LIN {X 0,Y 491.211,Z 1235.46,A -85,B 0,C 180,E1 12597.361,E2 12597.361} C_VEL
LIN {X 0,Y 492.197,Z 1227.239,A -85,B 0,C 180,E1 12605.326,E2 12605.326} C_VEL
LIN {X 0,Y 494.194,Z 1205.404,A -85,B 0,C 180,E1 12612.883,E2 12612.883} C_VEL
LIN {X 0,Y 499.705,Z 1169.344,A -85,B 0,C 180,E1 12619.985,E2 12619.985} C_VEL
LIN {X 0,Y 507.992,Z 1121.366,A -85,B 0,C 180,E1 12625.908,E2 12625.908} C_VEL
LIN {X 0,Y 516.438,Z 1064.19,A -85,B 0,C 180,E1 12630.398,E2 12630.398} C_VEL
LIN {X 0,Y 519.366,Z 1023.748,A -85,B 0,C 180,E1 12632.582,E2 12632.582} C_VEL
LIN {X 0,Y 493.539,Z 958.868,A -85,B 0,C 180,E1 12636.637,E2 12636.637} C_VEL
LIN {X 0,Y 489.609,Z 948.94,A -85,B 0,C 180,E1 12637.215,E2 12637.215} C_VEL
LIN {X 0,Y 489.5,Z 948.94,A -85,B 0,C 180,E1 12646.8,E2 12646.8} C_VEL
LIN {X 0,Y 489.694,Z 948.94,A -85,B 0,C 180,E1 12657.113,E2 12657.113} C_VEL
LIN {X 0,Y 490.223,Z 950.204,A -85,B 0,C 180,E1 12666.559,E2 12666.559} C_VEL
LIN {X 0,Y 504.518,Z 1001.153,A -85,B 0,C 180,E1 12668.035,E2 12668.035} C_VEL
LIN {X 0,Y 503.347,Z 1055.895,A -85,B 0,C 180,E1 12669.439,E2 12669.439} C_VEL
LIN {X 0,Y 500.138,Z 1101.192,A -85,B 0,C 180,E1 12672.409,E2 12672.409} C_VEL
LIN {X 0,Y 496.485,Z 1136.434,A -85,B 0,C 180,E1 12676.706,E2 12676.706} C_VEL
LIN {X 0,Y 493.765,Z 1159.555,A -85,B 0,C 180,E1 12682.008,E2 12682.008} C_VEL
LIN {X 0,Y 492.775,Z 1168.783,A -85,B 0,C 180,E1 12687.309,E2 12687.309} C_VEL
LIN {X 0,Y 492.851,Z 1166.502,A -85,B 0,C 180,E1 12692.603,E2 12692.603} C_VEL
LIN {X 0,Y 494.456,Z 1150.28,A -85,B 0,C 180,E1 12698.337,E2 12698.337} C_VEL
LIN {X 0,Y 497.549,Z 1121.567,A -85,B 0,C 180,E1 12703.177,E2 12703.177} C_VEL
LIN {X 0,Y 501.349,Z 1080.414,A -85,B 0,C 180,E1 12706.955,E2 12706.955} C_VEL
LIN {X 0,Y 503.697,Z 1033.18,A -85,B 0,C 180,E1 12709.116,E2 12709.116} C_VEL
LIN {X 0,Y 501.948,Z 988.132,A -85,B 0,C 180,E1 12709.997,E2 12709.997} C_VEL
LIN {X 0,Y 490.032,Z 948.94,A -85,B 0,C 180,E1 12711.337,E2 12711.337} C_VEL
LIN {X 0,Y 489.534,Z 948.94,A -85,B 0,C 180,E1 12721.467,E2 12721.467} C_VEL
LIN {X 0,Y 489.452,Z 948.94,A -85,B 0,C 180,E1 12731.738,E2 12731.738} C_VEL
LIN {X 0,Y 489.581,Z 948.94,A -85,B 0,C 180,E1 12740.517,E2 12740.517} C_VEL
LIN {X 0,Y 489.797,Z 948.94,A -85,B 0,C 180,E1 12749.229,E2 12749.229} C_VEL
LIN {X 0,Y 490.061,Z 948.94,A -85,B 0,C 180,E1 12759.116,E2 12759.116} C_VEL
LIN {X 0,Y 490.905,Z 948.94,A -85,B 0,C 180,E1 12768.389,E2 12768.389} C_VEL
LIN {X 0,Y 490.724,Z 948.94,A -85,B 0,C 180,E1 12779.097,E2 12779.097} C_VEL
LIN {X 0,Y 490.401,Z 948.94,A -85,B 0,C 180,E1 12787.988,E2 12787.988} C_VEL
LIN {X 0,Y 489.983,Z 948.94,A -85,B 0,C 180,E1 12797.096,E2 12797.096} C_VEL
LIN {X 0,Y 489.779,Z 948.94,A -85,B 0,C 180,E1 12806.682,E2 12806.682} C_VEL
LIN {X 0,Y 489.937,Z 948.94,A -85,B 0,C 180,E1 12814.947,E2 12814.947} C_VEL
LIN {X 0,Y 489.655,Z 948.94,A -85,B 0,C 180,E1 12824.198,E2 12824.198} C_VEL
LIN {X 0,Y 489.798,Z 950.405,A -85,B 0,C 180,E1 12826.839,E2 12826.839} C_VEL
LIN {X 0,Y 518.54,Z 1013.899,A -85,B 0,C 180,E1 12831.17,E2 12831.17} C_VEL
LIN {X 0,Y 525.213,Z 1042.25,A -85,B 0,C 180,E1 12832.797,E2 12832.797} C_VEL
LIN {X 0,Y 514.365,Z 1115.654,A -85,B 0,C 180,E1 12836.471,E2 12836.471} C_VEL
LIN {X 0,Y 504.365,Z 1179.97,A -85,B 0,C 180,E1 12841.767,E2 12841.767} C_VEL
LIN {X 0,Y 497.073,Z 1230.999,A -85,B 0,C 180,E1 12848.228,E2 12848.228} C_VEL
LIN {X 0,Y 492.921,Z 1267.707,A -85,B 0,C 180,E1 12855.512,E2 12855.512} C_VEL
LIN {X 0,Y 491.499,Z 1286.659,A -85,B 0,C 180,E1 12862.006,E2 12862.006} C_VEL
LIN {X 0,Y 483.413,Z 1292.195,A -85,B 0,C 180,E1 12866.028,E2 12866.028} C_VEL
LIN {X 0,Y 483.428,Z 1292.84,A -85,B 0,C 180,E1 12872.743,E2 12872.743} C_VEL
LIN {X 0,Y 483.602,Z 1280.706,A -85,B 0,C 180,E1 12879.619,E2 12879.619} C_VEL
LIN {X 0,Y 485.229,Z 1255.323,A -85,B 0,C 180,E1 12886.158,E2 12886.158} C_VEL
LIN {X 0,Y 488.81,Z 1214.714,A -85,B 0,C 180,E1 12892.396,E2 12892.396} C_VEL
LIN {X 0,Y 494.43,Z 1155.575,A -85,B 0,C 180,E1 12898.201,E2 12898.201} C_VEL
LIN {X 0,Y 502.044,Z 1074.735,A -85,B 0,C 180,E1 12903.395,E2 12903.395} C_VEL
LIN {X 0,Y 506.039,Z 1025.461,A -85,B 0,C 180,E1 12905.719,E2 12905.719} C_VEL
LIN {X 0,Y 497.61,Z 982.294,A -85,B 0,C 180,E1 12908.629,E2 12908.629} C_VEL
LIN {X 0,Y 488.368,Z 961.377,A -85,B 0,C 180,E1 12911.493,E2 12911.493} C_VEL
LIN {X 0,Y 485.546,Z 955.861,A -85,B 0,C 180,E1 12913.699,E2 12913.699} C_VEL
LIN {X 0,Y 487.532,Z 959.576,A -85,B 0,C 180,E1 12915.666,E2 12915.666} C_VEL
LIN {X 0,Y 497.122,Z 976.809,A -85,B 0,C 180,E1 12918.204,E2 12918.204} C_VEL
LIN {X 0,Y 509.017,Z 1015.646,A -85,B 0,C 180,E1 12920.57,E2 12920.57} C_VEL
LIN {X 0,Y 511.87,Z 1042.243,A -85,B 0,C 180,E1 12921.963,E2 12921.963} C_VEL
LIN {X 0,Y 505.638,Z 1098.199,A -85,B 0,C 180,E1 12925.235,E2 12925.235} C_VEL
LIN {X 0,Y 497.291,Z 1149.138,A -85,B 0,C 180,E1 12930.205,E2 12930.205} C_VEL
LIN {X 0,Y 489.898,Z 1189.814,A -85,B 0,C 180,E1 12936.565,E2 12936.565} C_VEL
LIN {X 0,Y 485.077,Z 1218.909,A -85,B 0,C 180,E1 12944.128,E2 12944.128} C_VEL
LIN {X 0,Y 483.428,Z 1233.639,A -85,B 0,C 180,E1 12951.896,E2 12951.896} C_VEL
LIN {X 0,Y 483.632,Z 1235.321,A -85,B 0,C 180,E1 12959.119,E2 12959.119} C_VEL
LIN {X 0,Y 484.255,Z 1225.816,A -85,B 0,C 180,E1 12966.316,E2 12966.316} C_VEL
LIN {X 0,Y 486.687,Z 1202.499,A -85,B 0,C 180,E1 12973.931,E2 12973.931} C_VEL
LIN {X 0,Y 492.837,Z 1165.138,A -85,B 0,C 180,E1 12980.997,E2 12980.997} C_VEL
LIN {X 0,Y 501.852,Z 1114.197,A -85,B 0,C 180,E1 12987.015,E2 12987.015} C_VEL
LIN {X 0,Y 510.637,Z 1055.281,A -85,B 0,C 180,E1 12991.363,E2 12991.363} C_VEL
LIN {X 0,Y 512.254,Z 1026.098,A -85,B 0,C 180,E1 12992.931,E2 12992.931} C_VEL
LIN {X 0,Y 486.656,Z 961.716,A -85,B 0,C 180,E1 12997.077,E2 12997.077} C_VEL
LIN {X 0,Y 481.499,Z 948.94,A -85,B 0,C 180,E1 12997.952,E2 12997.952} C_VEL
LIN {X 0,Y 481.524,Z 948.94,A -85,B 0,C 180,E1 13007.821,E2 13007.821} C_VEL
LIN {X 0,Y 481.663,Z 948.94,A -85,B 0,C 180,E1 13016.654,E2 13016.654} C_VEL
LIN {X 0,Y 482.137,Z 950.075,A -85,B 0,C 180,E1 13026.137,E2 13026.137} C_VEL
LIN {X 0,Y 497.113,Z 1003.116,A -85,B 0,C 180,E1 13027.718,E2 13027.718} C_VEL
LIN {X 0,Y 495.929,Z 1056.161,A -85,B 0,C 180,E1 13029.097,E2 13029.097} C_VEL
LIN {X 0,Y 492.737,Z 1100.792,A -85,B 0,C 180,E1 13032.02,E2 13032.02} C_VEL
LIN {X 0,Y 488.965,Z 1135.924,A -85,B 0,C 180,E1 13036.269,E2 13036.269} C_VEL
LIN {X 0,Y 486.183,Z 1159.161,A -85,B 0,C 180,E1 13041.431,E2 13041.431} C_VEL
LIN {X 0,Y 484.857,Z 1169.728,A -85,B 0,C 180,E1 13047.265,E2 13047.265} C_VEL
LIN {X 0,Y 484.934,Z 1167.468,A -85,B 0,C 180,E1 13052.646,E2 13052.646} C_VEL
LIN {X 0,Y 486.608,Z 1151.273,A -85,B 0,C 180,E1 13058.473,E2 13058.473} C_VEL
LIN {X 0,Y 489.828,Z 1122.592,A -85,B 0,C 180,E1 13063.388,E2 13063.388} C_VEL
LIN {X 0,Y 493.774,Z 1081.501,A -85,B 0,C 180,E1 13067.223,E2 13067.223} C_VEL
LIN {X 0,Y 496.241,Z 1033.419,A -85,B 0,C 180,E1 13069.445,E2 13069.445} C_VEL
LIN {X 0,Y 494.378,Z 989.209,A -85,B 0,C 180,E1 13070.324,E2 13070.324} C_VEL
LIN {X 0,Y 481.964,Z 948.94,A -85,B 0,C 180,E1 13071.67,E2 13071.67} C_VEL
LIN {X 0,Y 481.548,Z 948.94,A -85,B 0,C 180,E1 13081.272,E2 13081.272} C_VEL
LIN {X 0,Y 481.381,Z 948.94,A -85,B 0,C 180,E1 13090.193,E2 13090.193} C_VEL
LIN {X 0,Y 481.588,Z 948.94,A -85,B 0,C 180,E1 13100.453,E2 13100.453} C_VEL
LIN {X 0,Y 481.781,Z 948.94,A -85,B 0,C 180,E1 13110.75,E2 13110.75} C_VEL
LIN {X 0,Y 482.133,Z 948.94,A -85,B 0,C 180,E1 13120.679,E2 13120.679} C_VEL
LIN {X 0,Y 482.743,Z 948.94,A -85,B 0,C 180,E1 13130.024,E2 13130.024} C_VEL
LIN {X 0,Y 482.726,Z 948.94,A -85,B 0,C 180,E1 13139.082,E2 13139.082} C_VEL
LIN {X 0,Y 482.403,Z 948.94,A -85,B 0,C 180,E1 13148.122,E2 13148.122} C_VEL
LIN {X 0,Y 481.977,Z 948.94,A -85,B 0,C 180,E1 13157.389,E2 13157.389} C_VEL
LIN {X 0,Y 481.8,Z 948.94,A -85,B 0,C 180,E1 13167.16,E2 13167.16} C_VEL
LIN {X 0,Y 481.789,Z 948.94,A -85,B 0,C 180,E1 13176.652,E2 13176.652} C_VEL
LIN {X 0,Y 481.839,Z 950.706,A -85,B 0,C 180,E1 13186.117,E2 13186.117} C_VEL
LIN {X 0,Y 511.726,Z 1016.286,A -85,B 0,C 180,E1 13190.757,E2 13190.757} C_VEL
LIN {X 0,Y 518.055,Z 1044.204,A -85,B 0,C 180,E1 13192.418,E2 13192.418} C_VEL
LIN {X 0,Y 506.873,Z 1117.207,A -85,B 0,C 180,E1 13196.187,E2 13196.187} C_VEL
LIN {X 0,Y 496.491,Z 1181.713,A -85,B 0,C 180,E1 13201.66,E2 13201.66} C_VEL
LIN {X 0,Y 488.937,Z 1232.789,A -85,B 0,C 180,E1 13208.342,E2 13208.342} C_VEL
LIN {X 0,Y 484.766,Z 1268.623,A -85,B 0,C 180,E1 13215.741,E2 13215.741} C_VEL
LIN {X 0,Y 483.351,Z 1287.892,A -85,B 0,C 180,E1 13222.832,E2 13222.832} C_VEL
LIN {X 0,Y 483.413,Z 1292.195,A -85,B 0,C 180,E1 13226.028,E2 13226.028} C_VEL
LIN {X 0,Y 475.431,Z 1293.448,A -85,B 0,C 180,E1 13230.149,E2 13230.149} C_VEL
LIN {X 0,Y 475.669,Z 1285.828,A -85,B 0,C 180,E1 13237.376,E2 13237.376} C_VEL
LIN {X 0,Y 476.612,Z 1264.154,A -85,B 0,C 180,E1 13244.33,E2 13244.33} C_VEL
LIN {X 0,Y 479.603,Z 1228.689,A -85,B 0,C 180,E1 13250.722,E2 13250.722} C_VEL
LIN {X 0,Y 484.576,Z 1177.402,A -85,B 0,C 180,E1 13256.609,E2 13256.609} C_VEL
LIN {X 0,Y 492.062,Z 1103.72,A -85,B 0,C 180,E1 13262.17,E2 13262.17} C_VEL
LIN {X 0,Y 499.161,Z 1027.522,A -85,B 0,C 180,E1 13266.155,E2 13266.155} C_VEL
LIN {X 0,Y 492.068,Z 986.499,A -85,B 0,C 180,E1 13269.1,E2 13269.1} C_VEL
LIN {X 0,Y 484.839,Z 968.073,A -85,B 0,C 180,E1 13271.826,E2 13271.826} C_VEL
LIN {X 0,Y 483.253,Z 963.504,A -85,B 0,C 180,E1 13273.699,E2 13273.699} C_VEL
LIN {X 0,Y 485.534,Z 968.12,A -85,B 0,C 180,E1 13275.738,E2 13275.738} C_VEL
LIN {X 0,Y 494.868,Z 987.686,A -85,B 0,C 180,E1 13278.238,E2 13278.238} C_VEL
LIN {X 0,Y 505.961,Z 1038.4,A -85,B 0,C 180,E1 13281.22,E2 13281.22} C_VEL
LIN {X 0,Y 499.43,Z 1095.926,A -85,B 0,C 180,E1 13284.484,E2 13284.484} C_VEL
LIN {X 0,Y 490.562,Z 1148.251,A -85,B 0,C 180,E1 13289.555,E2 13289.555} C_VEL
LIN {X 0,Y 482.664,Z 1189.461,A -85,B 0,C 180,E1 13296.001,E2 13296.001} C_VEL
LIN {X 0,Y 477.603,Z 1218.168,A -85,B 0,C 180,E1 13303.399,E2 13303.399} C_VEL
LIN {X 0,Y 475.561,Z 1233.069,A -85,B 0,C 180,E1 13310.836,E2 13310.836} C_VEL
LIN {X 0,Y 475.656,Z 1235.818,A -85,B 0,C 180,E1 13319.104,E2 13319.104} C_VEL
LIN {X 0,Y 476.291,Z 1226.268,A -85,B 0,C 180,E1 13326.422,E2 13326.422} C_VEL
LIN {X 0,Y 478.805,Z 1203.262,A -85,B 0,C 180,E1 13334.059,E2 13334.059} C_VEL
LIN {X 0,Y 485.043,Z 1166.834,A -85,B 0,C 180,E1 13341.11,E2 13341.11} C_VEL
LIN {X 0,Y 494.309,Z 1116.083,A -85,B 0,C 180,E1 13347.252,E2 13347.252} C_VEL
LIN {X 0,Y 503.468,Z 1056.622,A -85,B 0,C 180,E1 13351.734,E2 13351.734} C_VEL
LIN {X 0,Y 504.78,Z 1027.337,A -85,B 0,C 180,E1 13353.364,E2 13353.364} C_VEL
LIN {X 0,Y 479.243,Z 962.842,A -85,B 0,C 180,E1 13357.605,E2 13357.605} C_VEL
LIN {X 0,Y 473.422,Z 948.94,A -85,B 0,C 180,E1 13358.489,E2 13358.489} C_VEL
LIN {X 0,Y 473.478,Z 948.94,A -85,B 0,C 180,E1 13368.907,E2 13368.907} C_VEL
LIN {X 0,Y 473.668,Z 948.94,A -85,B 0,C 180,E1 13378.154,E2 13378.154} C_VEL
LIN {X 0,Y 474.094,Z 950.032,A -85,B 0,C 180,E1 13385.703,E2 13385.703} C_VEL
LIN {X 0,Y 489.716,Z 1004.431,A -85,B 0,C 180,E1 13387.382,E2 13387.382} C_VEL
LIN {X 0,Y 488.405,Z 1058.374,A -85,B 0,C 180,E1 13388.833,E2 13388.833} C_VEL
LIN {X 0,Y 484.877,Z 1104.074,A -85,B 0,C 180,E1 13391.954,E2 13391.954} C_VEL
LIN {X 0,Y 480.827,Z 1139.501,A -85,B 0,C 180,E1 13396.497,E2 13396.497} C_VEL
LIN {X 0,Y 477.851,Z 1162.687,A -85,B 0,C 180,E1 13402.199,E2 13402.199} C_VEL
LIN {X 0,Y 476.943,Z 1170.672,A -85,B 0,C 180,E1 13407.22,E2 13407.22} C_VEL
LIN {X 0,Y 477.002,Z 1168.436,A -85,B 0,C 180,E1 13412.69,E2 13412.69} C_VEL
LIN {X 0,Y 478.771,Z 1152.266,A -85,B 0,C 180,E1 13418.612,E2 13418.612} C_VEL
LIN {X 0,Y 482.141,Z 1123.613,A -85,B 0,C 180,E1 13423.606,E2 13423.606} C_VEL
LIN {X 0,Y 486.231,Z 1082.61,A -85,B 0,C 180,E1 13427.497,E2 13427.497} C_VEL
LIN {X 0,Y 488.765,Z 1034.7,A -85,B 0,C 180,E1 13429.755,E2 13429.755} C_VEL
LIN {X 0,Y 486.955,Z 990.574,A -85,B 0,C 180,E1 13430.651,E2 13430.651} C_VEL
LIN {X 0,Y 473.877,Z 948.94,A -85,B 0,C 180,E1 13432.065,E2 13432.065} C_VEL
LIN {X 0,Y 473.483,Z 948.94,A -85,B 0,C 180,E1 13441.867,E2 13441.867} C_VEL
LIN {X 0,Y 473.35,Z 948.94,A -85,B 0,C 180,E1 13451.075,E2 13451.075} C_VEL
LIN {X 0,Y 473.552,Z 948.94,A -85,B 0,C 180,E1 13461.295,E2 13461.295} C_VEL
LIN {X 0,Y 473.738,Z 948.94,A -85,B 0,C 180,E1 13471.638,E2 13471.638} C_VEL
LIN {X 0,Y 474.228,Z 948.94,A -85,B 0,C 180,E1 13482.28,E2 13482.28} C_VEL
LIN {X 0,Y 474.739,Z 948.94,A -85,B 0,C 180,E1 13489.854,E2 13489.854} C_VEL
LIN {X 0,Y 474.729,Z 948.94,A -85,B 0,C 180,E1 13499.066,E2 13499.066} C_VEL
LIN {X 0,Y 474.38,Z 948.94,A -85,B 0,C 180,E1 13508.26,E2 13508.26} C_VEL
LIN {X 0,Y 473.937,Z 948.94,A -85,B 0,C 180,E1 13517.694,E2 13517.694} C_VEL
LIN {X 0,Y 473.793,Z 948.94,A -85,B 0,C 180,E1 13528.374,E2 13528.374} C_VEL
LIN {X 0,Y 473.776,Z 948.94,A -85,B 0,C 180,E1 13538.638,E2 13538.638} C_VEL
LIN {X 0,Y 473.693,Z 950.046,A -85,B 0,C 180,E1 13545.324,E2 13545.324} C_VEL
LIN {X 0,Y 504.735,Z 1018.436,A -85,B 0,C 180,E1 13550.321,E2 13550.321} C_VEL
LIN {X 0,Y 510.8,Z 1046.867,A -85,B 0,C 180,E1 13552.058,E2 13552.058} C_VEL
LIN {X 0,Y 499.452,Z 1117.969,A -85,B 0,C 180,E1 13555.857,E2 13555.857} C_VEL
LIN {X 0,Y 488.666,Z 1182.726,A -85,B 0,C 180,E1 13561.481,E2 13561.481} C_VEL
LIN {X 0,Y 480.986,Z 1233.279,A -85,B 0,C 180,E1 13568.256,E2 13568.256} C_VEL
LIN {X 0,Y 476.725,Z 1268.936,A -85,B 0,C 180,E1 13575.814,E2 13575.814} C_VEL
LIN {X 0,Y 475.384,Z 1287.302,A -85,B 0,C 180,E1 13582.711,E2 13582.711} C_VEL
LIN {X 0,Y 475.431,Z 1293.448,A -85,B 0,C 180,E1 13590.149,E2 13590.149} C_VEL
LIN {X 0,Y 467.315,Z 1290.285,A -85,B 0,C 180,E1 13594.35,E2 13594.35} C_VEL
LIN {X 0,Y 468.077,Z 1275.571,A -85,B 0,C 180,E1 13601.262,E2 13601.262} C_VEL
LIN {X 0,Y 470.614,Z 1244.576,A -85,B 0,C 180,E1 13608.369,E2 13608.369} C_VEL
LIN {X 0,Y 474.965,Z 1198.501,A -85,B 0,C 180,E1 13614.726,E2 13614.726} C_VEL
LIN {X 0,Y 481.596,Z 1133.866,A -85,B 0,C 180,E1 13620.543,E2 13620.543} C_VEL
LIN {X 0,Y 491.741,Z 1047.179,A -85,B 0,C 180,E1 13625.688,E2 13625.688} C_VEL
LIN {X 0,Y 491.841,Z 1025.815,A -85,B 0,C 180,E1 13626.899,E2 13626.899} C_VEL
LIN {X 0,Y 486.665,Z 990.335,A -85,B 0,C 180,E1 13629.65,E2 13629.65} C_VEL
LIN {X 0,Y 481.456,Z 974.599,A -85,B 0,C 180,E1 13632.223,E2 13632.223} C_VEL
LIN {X 0,Y 481.528,Z 971.562,A -85,B 0,C 180,E1 13634.562,E2 13634.562} C_VEL
LIN {X 0,Y 488.204,Z 987.393,A -85,B 0,C 180,E1 13637.276,E2 13637.276} C_VEL
LIN {X 0,Y 497.979,Z 1027.568,A -85,B 0,C 180,E1 13639.923,E2 13639.923} C_VEL
LIN {X 0,Y 498.576,Z 1052.151,A -85,B 0,C 180,E1 13641.223,E2 13641.223} C_VEL
LIN {X 0,Y 490.797,Z 1109.651,A -85,B 0,C 180,E1 13644.988,E2 13644.988} C_VEL
LIN {X 0,Y 481.538,Z 1158.317,A -85,B 0,C 180,E1 13650.292,E2 13650.292} C_VEL
LIN {X 0,Y 473.59,Z 1197.357,A -85,B 0,C 180,E1 13657.153,E2 13657.153} C_VEL
LIN {X 0,Y 468.851,Z 1223.639,A -85,B 0,C 180,E1 13665.009,E2 13665.009} C_VEL
LIN {X 0,Y 467.446,Z 1235.175,A -85,B 0,C 180,E1 13672.218,E2 13672.218} C_VEL
LIN {X 0,Y 467.659,Z 1236.315,A -85,B 0,C 180,E1 13679.088,E2 13679.088} C_VEL
LIN {X 0,Y 468.315,Z 1226.704,A -85,B 0,C 180,E1 13686.532,E2 13686.532} C_VEL
LIN {X 0,Y 470.986,Z 1203.576,A -85,B 0,C 180,E1 13694.297,E2 13694.297} C_VEL
LIN {X 0,Y 477.457,Z 1166.945,A -85,B 0,C 180,E1 13701.462,E2 13701.462} C_VEL
LIN {X 0,Y 487.048,Z 1116.162,A -85,B 0,C 180,E1 13707.663,E2 13707.663} C_VEL
LIN {X 0,Y 496.543,Z 1055.848,A -85,B 0,C 180,E1 13712.23,E2 13712.23} C_VEL
LIN {X 0,Y 497.927,Z 1030.54,A -85,B 0,C 180,E1 13713.661,E2 13713.661} C_VEL
LIN {X 0,Y 472.826,Z 966.515,A -85,B 0,C 180,E1 13718.003,E2 13718.003} C_VEL
LIN {X 0,Y 465.348,Z 948.94,A -85,B 0,C 180,E1 13719.074,E2 13719.074} C_VEL
LIN {X 0,Y 465.34,Z 948.94,A -85,B 0,C 180,E1 13727.993,E2 13727.993} C_VEL
LIN {X 0,Y 465.553,Z 948.94,A -85,B 0,C 180,E1 13737.415,E2 13737.415} C_VEL
LIN {X 0,Y 465.952,Z 949.108,A -85,B 0,C 180,E1 13745.232,E2 13745.232} C_VEL
LIN {X 0,Y 482.37,Z 1002.612,A -85,B 0,C 180,E1 13746.987,E2 13746.987} C_VEL
LIN {X 0,Y 481.055,Z 1058.272,A -85,B 0,C 180,E1 13748.454,E2 13748.454} C_VEL
LIN {X 0,Y 477.449,Z 1103.682,A -85,B 0,C 180,E1 13751.544,E2 13751.544} C_VEL
LIN {X 0,Y 473.333,Z 1139.095,A -85,B 0,C 180,E1 13756.042,E2 13756.042} C_VEL
LIN {X 0,Y 470.181,Z 1162.32,A -85,B 0,C 180,E1 13761.604,E2 13761.604} C_VEL
LIN {X 0,Y 469.025,Z 1171.617,A -85,B 0,C 180,E1 13767.173,E2 13767.173} C_VEL
LIN {X 0,Y 469.086,Z 1169.402,A -85,B 0,C 180,E1 13772.735,E2 13772.735} C_VEL
LIN {X 0,Y 470.946,Z 1153.257,A -85,B 0,C 180,E1 13778.757,E2 13778.757} C_VEL
LIN {X 0,Y 474.443,Z 1124.636,A -85,B 0,C 180,E1 13783.831,E2 13783.831} C_VEL
LIN {X 0,Y 478.687,Z 1083.694,A -85,B 0,C 180,E1 13787.782,E2 13787.782} C_VEL
LIN {X 0,Y 481.351,Z 1035.063,A -85,B 0,C 180,E1 13790.098,E2 13790.098} C_VEL
LIN {X 0,Y 479.674,Z 992.598,A -85,B 0,C 180,E1 13790.971,E2 13790.971} C_VEL
LIN {X 0,Y 465.838,Z 948.94,A -85,B 0,C 180,E1 13792.503,E2 13792.503} C_VEL
LIN {X 0,Y 465.388,Z 948.94,A -85,B 0,C 180,E1 13802.489,E2 13802.489} C_VEL
LIN {X 0,Y 465.323,Z 948.94,A -85,B 0,C 180,E1 13812.758,E2 13812.758} C_VEL
LIN {X 0,Y 465.521,Z 948.94,A -85,B 0,C 180,E1 13822.913,E2 13822.913} C_VEL
LIN {X 0,Y 465.751,Z 948.94,A -85,B 0,C 180,E1 13833.516,E2 13833.516} C_VEL
LIN {X 0,Y 466.428,Z 948.94,A -85,B 0,C 180,E1 13843.924,E2 13843.924} C_VEL
LIN {X 0,Y 466.414,Z 948.94,A -85,B 0,C 180,E1 13853.442,E2 13853.442} C_VEL
LIN {X 0,Y 466.568,Z 948.94,A -85,B 0,C 180,E1 13860.914,E2 13860.914} C_VEL
LIN {X 0,Y 466.293,Z 948.94,A -85,B 0,C 180,E1 13870.295,E2 13870.295} C_VEL
LIN {X 0,Y 465.85,Z 948.94,A -85,B 0,C 180,E1 13879.986,E2 13879.986} C_VEL
LIN {X 0,Y 465.812,Z 948.94,A -85,B 0,C 180,E1 13890.417,E2 13890.417} C_VEL
LIN {X 0,Y 465.612,Z 948.94,A -85,B 0,C 180,E1 13900.095,E2 13900.095} C_VEL
LIN {X 0,Y 465.859,Z 950.978,A -85,B 0,C 180,E1 13904.595,E2 13904.595} C_VEL
LIN {X 0,Y 497.47,Z 1019.856,A -85,B 0,C 180,E1 13909.836,E2 13909.836} C_VEL
LIN {X 0,Y 503.621,Z 1049.011,A -85,B 0,C 180,E1 13911.675,E2 13911.675} C_VEL
LIN {X 0,Y 491.73,Z 1120.498,A -85,B 0,C 180,E1 13915.648,E2 13915.648} C_VEL
LIN {X 0,Y 480.811,Z 1183.919,A -85,B 0,C 180,E1 13921.325,E2 13921.325} C_VEL
LIN {X 0,Y 472.99,Z 1234.05,A -85,B 0,C 180,E1 13928.227,E2 13928.227} C_VEL
LIN {X 0,Y 468.664,Z 1269.61,A -85,B 0,C 180,E1 13935.995,E2 13935.995} C_VEL
LIN {X 0,Y 467.324,Z 1288.245,A -85,B 0,C 180,E1 13943.521,E2 13943.521} C_VEL
LIN {X 0,Y 467.709,Z 1292.88,A -85,B 0,C 180,E1 13950.975,E2 13950.975} C_VEL
LIN {X 0,Y 467.315,Z 1290.285,A -85,B 0,C 180,E1 13954.35,E2 13954.35} C_VEL
LIN {X 0,Y 459.589,Z 1282.729,A -85,B 0,C 180,E1 13958.551,E2 13958.551} C_VEL
LIN {X 0,Y 460.933,Z 1259.457,A -85,B 0,C 180,E1 13965.561,E2 13965.561} C_VEL
LIN {X 0,Y 464.53,Z 1221.78,A -85,B 0,C 180,E1 13972.112,E2 13972.112} C_VEL
LIN {X 0,Y 470.574,Z 1165.89,A -85,B 0,C 180,E1 13978.318,E2 13978.318} C_VEL
LIN {X 0,Y 480.067,Z 1085.232,A -85,B 0,C 180,E1 13984.215,E2 13984.215} C_VEL
LIN {X 0,Y 485.802,Z 1030.749,A -85,B 0,C 180,E1 13987.213,E2 13987.213} C_VEL
LIN {X 0,Y 481.853,Z 995.487,A -85,B 0,C 180,E1 13990.092,E2 13990.092} C_VEL
LIN {X 0,Y 478.35,Z 979.934,A -85,B 0,C 180,E1 13993.058,E2 13993.058} C_VEL
LIN {X 0,Y 479.54,Z 981.557,A -85,B 0,C 180,E1 13994.971,E2 13994.971} C_VEL
LIN {X 0,Y 486.123,Z 999.348,A -85,B 0,C 180,E1 13997.4,E2 13997.4} C_VEL
LIN {X 0,Y 493.093,Z 1046.988,A -85,B 0,C 180,E1 14000.351,E2 14000.351} C_VEL
LIN {X 0,Y 485.494,Z 1103.489,A -85,B 0,C 180,E1 14003.858,E2 14003.858} C_VEL
LIN {X 0,Y 475.702,Z 1153.945,A -85,B 0,C 180,E1 14009.124,E2 14009.124} C_VEL
LIN {X 0,Y 467.052,Z 1193.721,A -85,B 0,C 180,E1 14015.824,E2 14015.824} C_VEL
LIN {X 0,Y 461.465,Z 1221.805,A -85,B 0,C 180,E1 14023.784,E2 14023.784} C_VEL
LIN {X 0,Y 459.577,Z 1235.227,A -85,B 0,C 180,E1 14031.472,E2 14031.472} C_VEL
LIN {X 0,Y 459.678,Z 1236.81,A -85,B 0,C 180,E1 14039.073,E2 14039.073} C_VEL
LIN {X 0,Y 460.372,Z 1226.184,A -85,B 0,C 180,E1 14047.121,E2 14047.121} C_VEL
LIN {X 0,Y 463.371,Z 1202.386,A -85,B 0,C 180,E1 14054.912,E2 14054.912} C_VEL
LIN {X 0,Y 470.154,Z 1165.495,A -85,B 0,C 180,E1 14062.054,E2 14062.054} C_VEL
LIN {X 0,Y 479.78,Z 1116.131,A -85,B 0,C 180,E1 14068.092,E2 14068.092} C_VEL
LIN {X 0,Y 489.396,Z 1056.98,A -85,B 0,C 180,E1 14072.627,E2 14072.627} C_VEL
LIN {X 0,Y 490.468,Z 1032.092,A -85,B 0,C 180,E1 14074.087,E2 14074.087} C_VEL
LIN {X 0,Y 465.279,Z 967.484,A -85,B 0,C 180,E1 14078.562,E2 14078.562} C_VEL
LIN {X 0,Y 457.271,Z 948.94,A -85,B 0,C 180,E1 14079.935,E2 14079.935} C_VEL
LIN {X 0,Y 457.359,Z 948.94,A -85,B 0,C 180,E1 14089.63,E2 14089.63} C_VEL
LIN {X 0,Y 457.55,Z 948.94,A -85,B 0,C 180,E1 14099.015,E2 14099.015} C_VEL
LIN {X 0,Y 457.993,Z 950.221,A -85,B 0,C 180,E1 14104.788,E2 14104.788} C_VEL
LIN {X 0,Y 475.014,Z 1003.297,A -85,B 0,C 180,E1 14106.618,E2 14106.618} C_VEL
LIN {X 0,Y 473.743,Z 1057.677,A -85,B 0,C 180,E1 14108.045,E2 14108.045} C_VEL
LIN {X 0,Y 470.114,Z 1103.282,A -85,B 0,C 180,E1 14111.123,E2 14111.123} C_VEL
LIN {X 0,Y 465.829,Z 1138.577,A -85,B 0,C 180,E1 14115.572,E2 14115.572} C_VEL
LIN {X 0,Y 462.617,Z 1161.99,A -85,B 0,C 180,E1 14121.015,E2 14121.015} C_VEL
LIN {X 0,Y 461.088,Z 1172.565,A -85,B 0,C 180,E1 14127.124,E2 14127.124} C_VEL
LIN {X 0,Y 461.182,Z 1170.365,A -85,B 0,C 180,E1 14132.782,E2 14132.782} C_VEL
LIN {X 0,Y 463.124,Z 1154.248,A -85,B 0,C 180,E1 14138.906,E2 14138.906} C_VEL
LIN {X 0,Y 466.772,Z 1125.656,A -85,B 0,C 180,E1 14144.063,E2 14144.063} C_VEL
LIN {X 0,Y 471.17,Z 1084.692,A -85,B 0,C 180,E1 14148.082,E2 14148.082} C_VEL
LIN {X 0,Y 473.921,Z 1036.351,A -85,B 0,C 180,E1 14150.427,E2 14150.427} C_VEL
LIN {X 0,Y 472.018,Z 993.132,A -85,B 0,C 180,E1 14151.345,E2 14151.345} C_VEL
LIN {X 0,Y 457.779,Z 948.94,A -85,B 0,C 180,E1 14152.955,E2 14152.955} C_VEL
LIN {X 0,Y 457.349,Z 948.94,A -85,B 0,C 180,E1 14163.132,E2 14163.132} C_VEL
LIN {X 0,Y 457.328,Z 948.94,A -85,B 0,C 180,E1 14172.789,E2 14172.789} C_VEL
LIN {X 0,Y 457.413,Z 948.94,A -85,B 0,C 180,E1 14182.106,E2 14182.106} C_VEL
LIN {X 0,Y 457.704,Z 948.94,A -85,B 0,C 180,E1 14191.359,E2 14191.359} C_VEL
LIN {X 0,Y 458.112,Z 948.94,A -85,B 0,C 180,E1 14201.635,E2 14201.635} C_VEL
LIN {X 0,Y 458.742,Z 948.94,A -85,B 0,C 180,E1 14209.496,E2 14209.496} C_VEL
LIN {X 0,Y 458.733,Z 948.94,A -85,B 0,C 180,E1 14219.034,E2 14219.034} C_VEL
LIN {X 0,Y 458.36,Z 948.94,A -85,B 0,C 180,E1 14228.551,E2 14228.551} C_VEL
LIN {X 0,Y 457.861,Z 948.94,A -85,B 0,C 180,E1 14238.337,E2 14238.337} C_VEL
LIN {X 0,Y 457.747,Z 948.94,A -85,B 0,C 180,E1 14248.716,E2 14248.716} C_VEL
LIN {X 0,Y 457.621,Z 948.94,A -85,B 0,C 180,E1 14258.892,E2 14258.892} C_VEL
LIN {X 0,Y 457.651,Z 950.426,A -85,B 0,C 180,E1 14263.761,E2 14263.761} C_VEL
LIN {X 0,Y 490.563,Z 1022.424,A -85,B 0,C 180,E1 14269.434,E2 14269.434} C_VEL
LIN {X 0,Y 496.519,Z 1050.691,A -85,B 0,C 180,E1 14271.267,E2 14271.267} C_VEL
LIN {X 0,Y 483.695,Z 1124.469,A -85,B 0,C 180,E1 14275.541,E2 14275.541} C_VEL
LIN {X 0,Y 472.63,Z 1187.1,A -85,B 0,C 180,E1 14281.397,E2 14281.397} C_VEL
LIN {X 0,Y 464.713,Z 1237.124,A -85,B 0,C 180,E1 14288.611,E2 14288.611} C_VEL
LIN {X 0,Y 460.472,Z 1270.969,A -85,B 0,C 180,E1 14296.423,E2 14296.423} C_VEL
LIN {X 0,Y 459.348,Z 1287.63,A -85,B 0,C 180,E1 14303.408,E2 14303.408} C_VEL
LIN {X 0,Y 459.723,Z 1292.376,A -85,B 0,C 180,E1 14310.992,E2 14310.992} C_VEL
LIN {X 0,Y 459.589,Z 1282.729,A -85,B 0,C 180,E1 14318.551,E2 14318.551} C_VEL
LIN {X 0,Y 452.516,Z 1271.023,A -85,B 0,C 180,E1 14322.678,E2 14322.678} C_VEL
LIN {X 0,Y 455.306,Z 1238.488,A -85,B 0,C 180,E1 14329.769,E2 14329.769} C_VEL
LIN {X 0,Y 460.577,Z 1189.684,A -85,B 0,C 180,E1 14336.313,E2 14336.313} C_VEL
LIN {X 0,Y 468.93,Z 1119.675,A -85,B 0,C 180,E1 14342.47,E2 14342.47} C_VEL
LIN {X 0,Y 479.653,Z 1033.664,A -85,B 0,C 180,E1 14347.711,E2 14347.711} C_VEL
LIN {X 0,Y 477.079,Z 999.349,A -85,B 0,C 180,E1 14350.749,E2 14350.749} C_VEL
LIN {X 0,Y 475.851,Z 987.226,A -85,B 0,C 180,E1 14353.34,E2 14353.34} C_VEL
LIN {X 0,Y 477.82,Z 991.282,A -85,B 0,C 180,E1 14355.305,E2 14355.305} C_VEL
LIN {X 0,Y 484.183,Z 1015.954,A -85,B 0,C 180,E1 14357.729,E2 14357.729} C_VEL
LIN {X 0,Y 486.779,Z 1052.082,A -85,B 0,C 180,E1 14359.92,E2 14359.92} C_VEL
LIN {X 0,Y 478.306,Z 1109.067,A -85,B 0,C 180,E1 14363.665,E2 14363.665} C_VEL
LIN {X 0,Y 467.716,Z 1159.37,A -85,B 0,C 180,E1 14369.226,E2 14369.226} C_VEL
LIN {X 0,Y 458.607,Z 1198.714,A -85,B 0,C 180,E1 14376.361,E2 14376.361} C_VEL
LIN {X 0,Y 453.182,Z 1224.837,A -85,B 0,C 180,E1 14384.478,E2 14384.478} C_VEL
LIN {X 0,Y 451.466,Z 1236.976,A -85,B 0,C 180,E1 14392.863,E2 14392.863} C_VEL
LIN {X 0,Y 451.551,Z 1235.953,A -85,B 0,C 180,E1 14400.982,E2 14400.982} C_VEL
LIN {X 0,Y 452.868,Z 1222.093,A -85,B 0,C 180,E1 14409.179,E2 14409.179} C_VEL
LIN {X 0,Y 457.552,Z 1193.138,A -85,B 0,C 180,E1 14417.39,E2 14417.39} C_VEL
LIN {X 0,Y 465.892,Z 1150.683,A -85,B 0,C 180,E1 14424.563,E2 14424.563} C_VEL
LIN {X 0,Y 476.28,Z 1095.323,A -85,B 0,C 180,E1 14430.403,E2 14430.403} C_VEL
LIN {X 0,Y 483.642,Z 1035.525,A -85,B 0,C 180,E1 14434.365,E2 14434.365} C_VEL
LIN {X 0,Y 458.994,Z 971.305,A -85,B 0,C 180,E1 14438.955,E2 14438.955} C_VEL
LIN {X 0,Y 449.236,Z 948.94,A -85,B 0,C 180,E1 14440.469,E2 14440.469} C_VEL
LIN {X 0,Y 449.417,Z 948.94,A -85,B 0,C 180,E1 14451.288,E2 14451.288} C_VEL
LIN {X 0,Y 449.55,Z 948.94,A -85,B 0,C 180,E1 14460.645,E2 14460.645} C_VEL
LIN {X 0,Y 450.014,Z 950.581,A -85,B 0,C 180,E1 14464.312,E2 14464.312} C_VEL
LIN {X 0,Y 467.688,Z 1007.564,A -85,B 0,C 180,E1 14466.297,E2 14466.297} C_VEL
LIN {X 0,Y 466.161,Z 1061.417,A -85,B 0,C 180,E1 14467.819,E2 14467.819} C_VEL
LIN {X 0,Y 462.281,Z 1106.566,A -85,B 0,C 180,E1 14471.039,E2 14471.039} C_VEL
LIN {X 0,Y 457.662,Z 1142.174,A -85,B 0,C 180,E1 14475.799,E2 14475.799} C_VEL
LIN {X 0,Y 454.26,Z 1165.454,A -85,B 0,C 180,E1 14481.791,E2 14481.791} C_VEL
LIN {X 0,Y 453.17,Z 1173.51,A -85,B 0,C 180,E1 14487.074,E2 14487.074} C_VEL
LIN {X 0,Y 453.265,Z 1171.33,A -85,B 0,C 180,E1 14492.831,E2 14492.831} C_VEL
LIN {X 0,Y 455.299,Z 1155.24,A -85,B 0,C 180,E1 14499.06,E2 14499.06} C_VEL
LIN {X 0,Y 459.098,Z 1126.677,A -85,B 0,C 180,E1 14504.303,E2 14504.303} C_VEL
LIN {X 0,Y 463.661,Z 1085.774,A -85,B 0,C 180,E1 14508.385,E2 14508.385} C_VEL
LIN {X 0,Y 466.455,Z 1038.598,A -85,B 0,C 180,E1 14510.737,E2 14510.737} C_VEL
LIN {X 0,Y 464.697,Z 994.711,A -85,B 0,C 180,E1 14511.697,E2 14511.697} C_VEL
LIN {X 0,Y 449.733,Z 948.94,A -85,B 0,C 180,E1 14513.535,E2 14513.535} C_VEL
LIN {X 0,Y 449.246,Z 948.94,A -85,B 0,C 180,E1 14524.098,E2 14524.098} C_VEL
LIN {X 0,Y 449.326,Z 948.94,A -85,B 0,C 180,E1 14533.741,E2 14533.741} C_VEL
LIN {X 0,Y 449.385,Z 948.94,A -85,B 0,C 180,E1 14543.744,E2 14543.744} C_VEL
LIN {X 0,Y 449.729,Z 948.94,A -85,B 0,C 180,E1 14553.279,E2 14553.279} C_VEL
LIN {X 0,Y 450.397,Z 948.94,A -85,B 0,C 180,E1 14563.588,E2 14563.588} C_VEL
LIN {X 0,Y 450.431,Z 948.94,A -85,B 0,C 180,E1 14573.208,E2 14573.208} C_VEL
LIN {X 0,Y 450.569,Z 948.94,A -85,B 0,C 180,E1 14580.946,E2 14580.946} C_VEL
LIN {X 0,Y 450.273,Z 948.94,A -85,B 0,C 180,E1 14590.665,E2 14590.665} C_VEL
LIN {X 0,Y 449.753,Z 948.94,A -85,B 0,C 180,E1 14600.733,E2 14600.733} C_VEL
LIN {X 0,Y 449.778,Z 948.94,A -85,B 0,C 180,E1 14611.515,E2 14611.515} C_VEL
LIN {X 0,Y 449.548,Z 948.94,A -85,B 0,C 180,E1 14621.151,E2 14621.151} C_VEL
LIN {X 0,Y 449.812,Z 950.97,A -85,B 0,C 180,E1 14622.979,E2 14622.979} C_VEL
LIN {X 0,Y 483.631,Z 1024.867,A -85,B 0,C 180,E1 14629.013,E2 14629.013} C_VEL
LIN {X 0,Y 489.454,Z 1051.815,A -85,B 0,C 180,E1 14630.844,E2 14630.844} C_VEL
LIN {X 0,Y 476.255,Z 1125.285,A -85,B 0,C 180,E1 14635.203,E2 14635.203} C_VEL
LIN {X 0,Y 464.722,Z 1188.374,A -85,B 0,C 180,E1 14641.265,E2 14641.265} C_VEL
LIN {X 0,Y 456.715,Z 1237.703,A -85,B 0,C 180,E1 14648.573,E2 14648.573} C_VEL
LIN {X 0,Y 452.435,Z 1271.131,A -85,B 0,C 180,E1 14656.498,E2 14656.498} C_VEL
LIN {X 0,Y 451.369,Z 1287,A -85,B 0,C 180,E1 14663.291,E2 14663.291} C_VEL
LIN {X 0,Y 451.728,Z 1291.874,A -85,B 0,C 180,E1 14671.01,E2 14671.01} C_VEL
LIN {X 0,Y 451.613,Z 1282.551,A -85,B 0,C 180,E1 14678.538,E2 14678.538} C_VEL
LIN {X 0,Y 452.516,Z 1271.023,A -85,B 0,C 180,E1 14682.678,E2 14682.678} C_VEL
LIN {X 0,Y 445.459,Z 1255.687,A -85,B 0,C 180,E1 14686.664,E2 14686.664} C_VEL
LIN {X 0,Y 449.726,Z 1216.337,A -85,B 0,C 180,E1 14693.404,E2 14693.404} C_VEL
LIN {X 0,Y 457.061,Z 1157.057,A -85,B 0,C 180,E1 14699.947,E2 14699.947} C_VEL
LIN {X 0,Y 469.177,Z 1070.702,A -85,B 0,C 180,E1 14706.258,E2 14706.258} C_VEL
LIN {X 0,Y 473.757,Z 1035.97,A -85,B 0,C 180,E1 14708.316,E2 14708.316} C_VEL
LIN {X 0,Y 473.082,Z 1005.386,A -85,B 0,C 180,E1 14711.168,E2 14711.168} C_VEL
LIN {X 0,Y 473.497,Z 994.773,A -85,B 0,C 180,E1 14713.609,E2 14713.609} C_VEL
LIN {X 0,Y 475.858,Z 1002.415,A -85,B 0,C 180,E1 14715.598,E2 14715.598} C_VEL
LIN {X 0,Y 481.938,Z 1045.885,A -85,B 0,C 180,E1 14718.924,E2 14718.924} C_VEL
LIN {X 0,Y 473.369,Z 1103.341,A -85,B 0,C 180,E1 14722.49,E2 14722.49} C_VEL
LIN {X 0,Y 462.55,Z 1153.614,A -85,B 0,C 180,E1 14727.798,E2 14727.798} C_VEL
LIN {X 0,Y 452.93,Z 1193.07,A -85,B 0,C 180,E1 14734.507,E2 14734.507} C_VEL
LIN {X 0,Y 446.442,Z 1221.414,A -85,B 0,C 180,E1 14742.534,E2 14742.534} C_VEL
LIN {X 0,Y 443.702,Z 1236.349,A -85,B 0,C 180,E1 14751.164,E2 14751.164} C_VEL
LIN {X 0,Y 443.682,Z 1237.8,A -85,B 0,C 180,E1 14759.039,E2 14759.039} C_VEL
LIN {X 0,Y 444.489,Z 1226.865,A -85,B 0,C 180,E1 14767.438,E2 14767.438} C_VEL
LIN {X 0,Y 448.008,Z 1201.694,A -85,B 0,C 180,E1 14775.745,E2 14775.745} C_VEL
LIN {X 0,Y 455.745,Z 1162.841,A -85,B 0,C 180,E1 14783.228,E2 14783.228} C_VEL
LIN {X 0,Y 466.099,Z 1111.724,A -85,B 0,C 180,E1 14789.394,E2 14789.394} C_VEL
LIN {X 0,Y 476.296,Z 1050.96,A -85,B 0,C 180,E1 14793.916,E2 14793.916} C_VEL
LIN {X 0,Y 475.749,Z 1035.67,A -85,B 0,C 180,E1 14794.914,E2 14794.914} C_VEL
LIN {X 0,Y 451.173,Z 971.799,A -85,B 0,C 180,E1 14799.574,E2 14799.574} C_VEL
LIN {X 0,Y 441.232,Z 948.94,A -85,B 0,C 180,E1 14801.156,E2 14801.156} C_VEL
LIN {X 0,Y 441.358,Z 948.94,A -85,B 0,C 180,E1 14810.723,E2 14810.723} C_VEL
LIN {X 0,Y 441.525,Z 948.94,A -85,B 0,C 180,E1 14821.275,E2 14821.275} C_VEL
LIN {X 0,Y 441.948,Z 950.552,A -85,B 0,C 180,E1 14823.804,E2 14823.804} C_VEL
LIN {X 0,Y 460.376,Z 1007.053,A -85,B 0,C 180,E1 14825.886,E2 14825.886} C_VEL
LIN {X 0,Y 458.886,Z 1060.943,A -85,B 0,C 180,E1 14827.387,E2 14827.387} C_VEL
LIN {X 0,Y 454.882,Z 1106.177,A -85,B 0,C 180,E1 14830.592,E2 14830.592} C_VEL
LIN {X 0,Y 450.24,Z 1141.755,A -85,B 0,C 180,E1 14835.311,E2 14835.311} C_VEL
LIN {X 0,Y 446.652,Z 1165.082,A -85,B 0,C 180,E1 14841.158,E2 14841.158} C_VEL
LIN {X 0,Y 445.264,Z 1174.454,A -85,B 0,C 180,E1 14847.022,E2 14847.022} C_VEL
LIN {X 0,Y 445.347,Z 1172.295,A -85,B 0,C 180,E1 14852.881,E2 14852.881} C_VEL
LIN {X 0,Y 447.471,Z 1156.232,A -85,B 0,C 180,E1 14859.22,E2 14859.22} C_VEL
LIN {X 0,Y 451.425,Z 1127.699,A -85,B 0,C 180,E1 14864.551,E2 14864.551} C_VEL
LIN {X 0,Y 456.097,Z 1087.851,A -85,B 0,C 180,E1 14868.625,E2 14868.625} C_VEL
LIN {X 0,Y 459.039,Z 1039.882,A -85,B 0,C 180,E1 14871.086,E2 14871.086} C_VEL
LIN {X 0,Y 457.427,Z 996.512,A -85,B 0,C 180,E1 14872.055,E2 14872.055} C_VEL
LIN {X 0,Y 441.664,Z 948.94,A -85,B 0,C 180,E1 14874.024,E2 14874.024} C_VEL
LIN {X 0,Y 441.204,Z 948.94,A -85,B 0,C 180,E1 14884.512,E2 14884.512} C_VEL
LIN {X 0,Y 441.269,Z 948.94,A -85,B 0,C 180,E1 14895.133,E2 14895.133} C_VEL
LIN {X 0,Y 441.422,Z 948.94,A -85,B 0,C 180,E1 14905.411,E2 14905.411} C_VEL
LIN {X 0,Y 441.735,Z 948.94,A -85,B 0,C 180,E1 14915.418,E2 14915.418} C_VEL
LIN {X 0,Y 442.512,Z 948.94,A -85,B 0,C 180,E1 14925.073,E2 14925.073} C_VEL
LIN {X 0,Y 442.679,Z 948.94,A -85,B 0,C 180,E1 14935.063,E2 14935.063} C_VEL
LIN {X 0,Y 442.814,Z 948.94,A -85,B 0,C 180,E1 14944.896,E2 14944.896} C_VEL
LIN {X 0,Y 442.067,Z 948.94,A -85,B 0,C 180,E1 14954.902,E2 14954.902} C_VEL
LIN {X 0,Y 441.622,Z 948.94,A -85,B 0,C 180,E1 14965.421,E2 14965.421} C_VEL
LIN {X 0,Y 441.683,Z 948.94,A -85,B 0,C 180,E1 14976.252,E2 14976.252} C_VEL
LIN {X 0,Y 441.713,Z 950.767,A -85,B 0,C 180,E1 14982.12,E2 14982.12} C_VEL
LIN {X 0,Y 476.182,Z 1025.849,A -85,B 0,C 180,E1 14988.481,E2 14988.481} C_VEL
LIN {X 0,Y 482.252,Z 1053.634,A -85,B 0,C 180,E1 14990.444,E2 14990.444} C_VEL
LIN {X 0,Y 468.833,Z 1125.928,A -85,B 0,C 180,E1 14994.854,E2 14994.854} C_VEL
LIN {X 0,Y 456.809,Z 1189.612,A -85,B 0,C 180,E1 15001.127,E2 15001.127} C_VEL
LIN {X 0,Y 448.741,Z 1238.092,A -85,B 0,C 180,E1 15008.505,E2 15008.505} C_VEL
LIN {X 0,Y 444.619,Z 1269.603,A -85,B 0,C 180,E1 15016.05,E2 15016.05} C_VEL
LIN {X 0,Y 443.408,Z 1286.359,A -85,B 0,C 180,E1 15023.17,E2 15023.17} C_VEL
LIN {X 0,Y 443.307,Z 1291.447,A -85,B 0,C 180,E1 15029.068,E2 15029.068} C_VEL
LIN {X 0,Y 443.575,Z 1287.075,A -85,B 0,C 180,E1 15035.938,E2 15035.938} C_VEL
LIN {X 0,Y 444.63,Z 1268.555,A -85,B 0,C 180,E1 15043.455,E2 15043.455} C_VEL
LIN {X 0,Y 445.459,Z 1255.687,A -85,B 0,C 180,E1 15046.664,E2 15046.664} C_VEL
LIN {X 0,Y 439.739,Z 1236.966,A -85,B 0,C 180,E1 15050.517,E2 15050.517} C_VEL
LIN {X 0,Y 445.877,Z 1186.931,A -85,B 0,C 180,E1 15057.402,E2 15057.402} C_VEL
LIN {X 0,Y 456.386,Z 1113.079,A -85,B 0,C 180,E1 15064.086,E2 15064.086} C_VEL
LIN {X 0,Y 468.219,Z 1037.58,A -85,B 0,C 180,E1 15069.051,E2 15069.051} C_VEL
LIN {X 0,Y 469.476,Z 1009.968,A -85,B 0,C 180,E1 15071.869,E2 15071.869} C_VEL
LIN {X 0,Y 471.496,Z 1002.921,A -85,B 0,C 180,E1 15074.086,E2 15074.086} C_VEL
LIN {X 0,Y 474.281,Z 1021.078,A -85,B 0,C 180,E1 15076.33,E2 15076.33} C_VEL
LIN {X 0,Y 475.136,Z 1058.027,A -85,B 0,C 180,E1 15078.769,E2 15078.769} C_VEL
LIN {X 0,Y 465.141,Z 1114.873,A -85,B 0,C 180,E1 15082.762,E2 15082.762} C_VEL
LIN {X 0,Y 453.453,Z 1163.427,A -85,B 0,C 180,E1 15088.488,E2 15088.488} C_VEL
LIN {X 0,Y 443.45,Z 1201.445,A -85,B 0,C 180,E1 15095.807,E2 15095.807} C_VEL
LIN {X 0,Y 437.623,Z 1226.15,A -85,B 0,C 180,E1 15103.911,E2 15103.911} C_VEL
LIN {X 0,Y 435.759,Z 1236.933,A -85,B 0,C 180,E1 15111.002,E2 15111.002} C_VEL
LIN {X 0,Y 435.684,Z 1238.292,A -85,B 0,C 180,E1 15119.021,E2 15119.021} C_VEL
LIN {X 0,Y 436.532,Z 1227.381,A -85,B 0,C 180,E1 15127.502,E2 15127.502} C_VEL
LIN {X 0,Y 439.854,Z 1203.799,A -85,B 0,C 180,E1 15135.531,E2 15135.531} C_VEL
LIN {X 0,Y 447.345,Z 1166.898,A -85,B 0,C 180,E1 15142.987,E2 15142.987} C_VEL
LIN {X 0,Y 457.863,Z 1117.267,A -85,B 0,C 180,E1 15149.294,E2 15149.294} C_VEL
LIN {X 0,Y 468.419,Z 1057.479,A -85,B 0,C 180,E1 15154.018,E2 15154.018} C_VEL
LIN {X 0,Y 469.075,Z 1039.571,A -85,B 0,C 180,E1 15155.155,E2 15155.155} C_VEL
LIN {X 0,Y 445.408,Z 976.854,A -85,B 0,C 180,E1 15159.888,E2 15159.888} C_VEL
LIN {X 0,Y 433.171,Z 948.94,A -85,B 0,C 180,E1 15161.888,E2 15161.888} C_VEL
LIN {X 0,Y 433.289,Z 948.94,A -85,B 0,C 180,E1 15172.145,E2 15172.145} C_VEL
LIN {X 0,Y 433.88,Z 950.486,A -85,B 0,C 180,E1 15183.275,E2 15183.275} C_VEL
LIN {X 0,Y 453.106,Z 1009.305,A -85,B 0,C 180,E1 15185.51,E2 15185.51} C_VEL
LIN {X 0,Y 451.453,Z 1063.029,A -85,B 0,C 180,E1 15187.066,E2 15187.066} C_VEL
LIN {X 0,Y 447.272,Z 1108.231,A -85,B 0,C 180,E1 15190.377,E2 15190.377} C_VEL
LIN {X 0,Y 442.278,Z 1143.956,A -85,B 0,C 180,E1 15195.294,E2 15195.294} C_VEL
LIN {X 0,Y 438.578,Z 1167.294,A -85,B 0,C 180,E1 15201.496,E2 15201.496} C_VEL
LIN {X 0,Y 437.346,Z 1175.399,A -85,B 0,C 180,E1 15206.968,E2 15206.968} C_VEL
LIN {X 0,Y 437.431,Z 1173.26,A -85,B 0,C 180,E1 15212.933,E2 15212.933} C_VEL
LIN {X 0,Y 439.565,Z 1157.736,A -85,B 0,C 180,E1 15219.251,E2 15219.251} C_VEL
LIN {X 0,Y 443.757,Z 1128.721,A -85,B 0,C 180,E1 15224.809,E2 15224.809} C_VEL
LIN {X 0,Y 448.614,Z 1088.932,A -85,B 0,C 180,E1 15228.947,E2 15228.947} C_VEL
LIN {X 0,Y 451.679,Z 1040.443,A -85,B 0,C 180,E1 15231.47,E2 15231.47} C_VEL
LIN {X 0,Y 449.895,Z 997.528,A -85,B 0,C 180,E1 15232.454,E2 15232.454} C_VEL
LIN {X 0,Y 433.613,Z 948.94,A -85,B 0,C 180,E1 15234.534,E2 15234.534} C_VEL
LIN {X 0,Y 433.178,Z 948.94,A -85,B 0,C 180,E1 15245.245,E2 15245.245} C_VEL
LIN {X 0,Y 433.22,Z 948.94,A -85,B 0,C 180,E1 15255.816,E2 15255.816} C_VEL
LIN {X 0,Y 433.41,Z 948.94,A -85,B 0,C 180,E1 15265.267,E2 15265.267} C_VEL
LIN {X 0,Y 433.73,Z 948.94,A -85,B 0,C 180,E1 15276.248,E2 15276.248} C_VEL
LIN {X 0,Y 434.682,Z 948.94,A -85,B 0,C 180,E1 15286.861,E2 15286.861} C_VEL
LIN {X 0,Y 435.046,Z 948.94,A -85,B 0,C 180,E1 15297.011,E2 15297.011} C_VEL
LIN {X 0,Y 434.555,Z 948.94,A -85,B 0,C 180,E1 15307.002,E2 15307.002} C_VEL
LIN {X 0,Y 433.833,Z 948.94,A -85,B 0,C 180,E1 15317.28,E2 15317.28} C_VEL
LIN {X 0,Y 433.602,Z 948.94,A -85,B 0,C 180,E1 15328.178,E2 15328.178} C_VEL
LIN {X 0,Y 433.492,Z 948.94,A -85,B 0,C 180,E1 15338.126,E2 15338.126} C_VEL
LIN {X 0,Y 433.733,Z 950.736,A -85,B 0,C 180,E1 15341.257,E2 15341.257} C_VEL
LIN {X 0,Y 469.335,Z 1028.495,A -85,B 0,C 180,E1 15348.065,E2 15348.065} C_VEL
LIN {X 0,Y 475.007,Z 1055.658,A -85,B 0,C 180,E1 15350.049,E2 15350.049} C_VEL
LIN {X 0,Y 461.12,Z 1127.872,A -85,B 0,C 180,E1 15354.611,E2 15354.611} C_VEL
LIN {X 0,Y 448.966,Z 1190.472,A -85,B 0,C 180,E1 15360.945,E2 15360.945} C_VEL
LIN {X 0,Y 440.584,Z 1239.463,A -85,B 0,C 180,E1 15368.629,E2 15368.629} C_VEL
LIN {X 0,Y 436.46,Z 1270.708,A -85,B 0,C 180,E1 15376.436,E2 15376.436} C_VEL
LIN {X 0,Y 435.466,Z 1287.272,A -85,B 0,C 180,E1 15384.159,E2 15384.159} C_VEL
LIN {X 0,Y 435.738,Z 1290.867,A -85,B 0,C 180,E1 15391.047,E2 15391.047} C_VEL
LIN {X 0,Y 435.624,Z 1282.159,A -85,B 0,C 180,E1 15398.562,E2 15398.562} C_VEL
LIN {X 0,Y 437.105,Z 1259.64,A -85,B 0,C 180,E1 15405.915,E2 15405.915} C_VEL
LIN {X 0,Y 439.739,Z 1236.966,A -85,B 0,C 180,E1 15410.517,E2 15410.517} C_VEL
LIN {X 0,Y 434.588,Z 1215.734,A -85,B 0,C 180,E1 15414.18,E2 15414.18} C_VEL
LIN {X 0,Y 443.179,Z 1155.528,A -85,B 0,C 180,E1 15421.131,E2 15421.131} C_VEL
LIN {X 0,Y 458.616,Z 1067.891,A -85,B 0,C 180,E1 15427.891,E2 15427.891} C_VEL
LIN {X 0,Y 463.347,Z 1039.385,A -85,B 0,C 180,E1 15429.86,E2 15429.86} C_VEL
LIN {X 0,Y 466.66,Z 1015.43,A -85,B 0,C 180,E1 15432.501,E2 15432.501} C_VEL
LIN {X 0,Y 469.007,Z 1011.422,A -85,B 0,C 180,E1 15434.134,E2 15434.134} C_VEL
LIN {X 0,Y 470.586,Z 1039.711,A -85,B 0,C 180,E1 15436.747,E2 15436.747} C_VEL
LIN {X 0,Y 468.062,Z 1070.828,A -85,B 0,C 180,E1 15438.704,E2 15438.704} C_VEL
LIN {X 0,Y 456.851,Z 1126.009,A -85,B 0,C 180,E1 15443.1,E2 15443.1} C_VEL
LIN {X 0,Y 444.18,Z 1173.332,A -85,B 0,C 180,E1 15449.354,E2 15449.354} C_VEL
LIN {X 0,Y 434.473,Z 1208.001,A -85,B 0,C 180,E1 15456.88,E2 15456.88} C_VEL
LIN {X 0,Y 429.052,Z 1230.817,A -85,B 0,C 180,E1 15465.683,E2 15465.683} C_VEL
LIN {X 0,Y 427.564,Z 1238.901,A -85,B 0,C 180,E1 15472.883,E2 15472.883} C_VEL
LIN {X 0,Y 427.598,Z 1237.355,A -85,B 0,C 180,E1 15481.037,E2 15481.037} C_VEL
LIN {X 0,Y 429.139,Z 1223.052,A -85,B 0,C 180,E1 15489.692,E2 15489.692} C_VEL
LIN {X 0,Y 434.514,Z 1193.454,A -85,B 0,C 180,E1 15498.344,E2 15498.344} C_VEL
LIN {X 0,Y 443.408,Z 1151.911,A -85,B 0,C 180,E1 15505.626,E2 15505.626} C_VEL
LIN {X 0,Y 454.646,Z 1096.808,A -85,B 0,C 180,E1 15511.661,E2 15511.661} C_VEL
LIN {X 0,Y 462.208,Z 1042.963,A -85,B 0,C 180,E1 15515.438,E2 15515.438} C_VEL
LIN {X 0,Y 439.077,Z 980.638,A -85,B 0,C 180,E1 15520.293,E2 15520.293} C_VEL
LIN {X 0,Y 425.102,Z 948.94,A -85,B 0,C 180,E1 15522.898,E2 15522.898} C_VEL
LIN {X 0,Y 425.233,Z 948.94,A -85,B 0,C 180,E1 15533.87,E2 15533.87} C_VEL
LIN {X 0,Y 425.87,Z 950.714,A -85,B 0,C 180,E1 15542.732,E2 15542.732} C_VEL
LIN {X 0,Y 445.836,Z 1009.938,A -85,B 0,C 180,E1 15545.092,E2 15545.092} C_VEL
LIN {X 0,Y 444.124,Z 1063.927,A -85,B 0,C 180,E1 15546.676,E2 15546.676} C_VEL
LIN {X 0,Y 439.774,Z 1109.066,A -85,B 0,C 180,E1 15550.029,E2 15550.029} C_VEL
LIN {X 0,Y 434.611,Z 1144.846,A -85,B 0,C 180,E1 15555.029,E2 15555.029} C_VEL
LIN {X 0,Y 430.726,Z 1168.216,A -85,B 0,C 180,E1 15561.34,E2 15561.34} C_VEL
LIN {X 0,Y 429.438,Z 1176.343,A -85,B 0,C 180,E1 15566.912,E2 15566.912} C_VEL
LIN {X 0,Y 429.516,Z 1174.224,A -85,B 0,C 180,E1 15572.987,E2 15572.987} C_VEL
LIN {X 0,Y 431.733,Z 1158.729,A -85,B 0,C 180,E1 15579.42,E2 15579.42} C_VEL
LIN {X 0,Y 436.11,Z 1129.741,A -85,B 0,C 180,E1 15585.074,E2 15585.074} C_VEL
LIN {X 0,Y 441.138,Z 1090.013,A -85,B 0,C 180,E1 15589.281,E2 15589.281} C_VEL
LIN {X 0,Y 444.336,Z 1041.674,A -85,B 0,C 180,E1 15591.843,E2 15591.843} C_VEL
LIN {X 0,Y 442.635,Z 999.305,A -85,B 0,C 180,E1 15592.838,E2 15592.838} C_VEL
LIN {X 0,Y 425.535,Z 948.94,A -85,B 0,C 180,E1 15594.995,E2 15594.995} C_VEL
LIN {X 0,Y 425.069,Z 948.94,A -85,B 0,C 180,E1 15606.021,E2 15606.021} C_VEL
LIN {X 0,Y 425.223,Z 948.94,A -85,B 0,C 180,E1 15616.936,E2 15616.936} C_VEL
LIN {X 0,Y 425.436,Z 948.94,A -85,B 0,C 180,E1 15626.848,E2 15626.848} C_VEL
LIN {X 0,Y 425.786,Z 948.94,A -85,B 0,C 180,E1 15637.998,E2 15637.998} C_VEL
LIN {X 0,Y 426.693,Z 948.94,A -85,B 0,C 180,E1 15648.697,E2 15648.697} C_VEL
LIN {X 0,Y 426.78,Z 948.94,A -85,B 0,C 180,E1 15658.961,E2 15658.961} C_VEL
LIN {X 0,Y 426.274,Z 948.94,A -85,B 0,C 180,E1 15669.2,E2 15669.2} C_VEL
LIN {X 0,Y 425.704,Z 948.94,A -85,B 0,C 180,E1 15679.777,E2 15679.777} C_VEL
LIN {X 0,Y 425.597,Z 948.94,A -85,B 0,C 180,E1 15691.115,E2 15691.115} C_VEL
LIN {X 0,Y 425.677,Z 950.21,A -85,B 0,C 180,E1 15700.341,E2 15700.341} C_VEL
LIN {X 0,Y 462.185,Z 1030.44,A -85,B 0,C 180,E1 15707.61,E2 15707.61} C_VEL
LIN {X 0,Y 467.893,Z 1056.933,A -85,B 0,C 180,E1 15709.61,E2 15709.61} C_VEL
LIN {X 0,Y 453.499,Z 1129.354,A -85,B 0,C 180,E1 15714.331,E2 15714.331} C_VEL
LIN {X 0,Y 441.127,Z 1191.308,A -85,B 0,C 180,E1 15720.769,E2 15720.769} C_VEL
LIN {X 0,Y 432.688,Z 1239.253,A -85,B 0,C 180,E1 15728.449,E2 15728.449} C_VEL
LIN {X 0,Y 428.38,Z 1271.413,A -85,B 0,C 180,E1 15736.741,E2 15736.741} C_VEL
LIN {X 0,Y 427.512,Z 1286.844,A -85,B 0,C 180,E1 15744.218,E2 15744.218} C_VEL
LIN {X 0,Y 427.756,Z 1290.364,A -85,B 0,C 180,E1 15751.066,E2 15751.066} C_VEL
LIN {X 0,Y 427.648,Z 1281.677,A -85,B 0,C 180,E1 15758.723,E2 15758.723} C_VEL
LIN {X 0,Y 429.123,Z 1260.12,A -85,B 0,C 180,E1 15765.956,E2 15765.956} C_VEL
LIN {X 0,Y 433.346,Z 1223.855,A -85,B 0,C 180,E1 15772.978,E2 15772.978} C_VEL
LIN {X 0,Y 434.588,Z 1215.734,A -85,B 0,C 180,E1 15774.18,E2 15774.18} C_VEL
LIN {X 0,Y 430.545,Z 1192.478,A -85,B 0,C 180,E1 15777.697,E2 15777.697} C_VEL
LIN {X 0,Y 443.459,Z 1117.067,A -85,B 0,C 180,E1 15785.175,E2 15785.175} C_VEL
LIN {X 0,Y 459.131,Z 1043.536,A -85,B 0,C 180,E1 15790.525,E2 15790.525} C_VEL
LIN {X 0,Y 464.543,Z 1021.47,A -85,B 0,C 180,E1 15793.09,E2 15793.09} C_VEL
LIN {X 0,Y 466.127,Z 1020.705,A -85,B 0,C 180,E1 15794.089,E2 15794.089} C_VEL
LIN {X 0,Y 464.724,Z 1062.149,A -85,B 0,C 180,E1 15797.38,E2 15797.38} C_VEL
LIN {X 0,Y 452.622,Z 1119.934,A -85,B 0,C 180,E1 15801.681,E2 15801.681} C_VEL
LIN {X 0,Y 439.158,Z 1168.581,A -85,B 0,C 180,E1 15807.823,E2 15807.823} C_VEL
LIN {X 0,Y 428.023,Z 1205.618,A -85,B 0,C 180,E1 15815.54,E2 15815.54} C_VEL
LIN {X 0,Y 421.546,Z 1229.63,A -85,B 0,C 180,E1 15824.354,E2 15824.354} C_VEL
LIN {X 0,Y 419.612,Z 1239.478,A -85,B 0,C 180,E1 15832.747,E2 15832.747} C_VEL
LIN {X 0,Y 419.611,Z 1237.815,A -85,B 0,C 180,E1 15841.057,E2 15841.057} C_VEL
LIN {X 0,Y 421.004,Z 1224.63,A -85,B 0,C 180,E1 15849.357,E2 15849.357} C_VEL
LIN {X 0,Y 426.297,Z 1195.797,A -85,B 0,C 180,E1 15858.173,E2 15858.173} C_VEL
LIN {X 0,Y 435.657,Z 1153.384,A -85,B 0,C 180,E1 15865.838,E2 15865.838} C_VEL
LIN {X 0,Y 447.052,Z 1099.219,A -85,B 0,C 180,E1 15871.935,E2 15871.935} C_VEL
LIN {X 0,Y 454.897,Z 1045.014,A -85,B 0,C 180,E1 15875.844,E2 15875.844} C_VEL
LIN {X 0,Y 432.436,Z 983.916,A -85,B 0,C 180,E1 15880.744,E2 15880.744} C_VEL
LIN {X 0,Y 417.078,Z 948.94,A -85,B 0,C 180,E1 15883.454,E2 15883.454} C_VEL
LIN {X 0,Y 417.195,Z 948.94,A -85,B 0,C 180,E1 15893.06,E2 15893.06} C_VEL
LIN {X 0,Y 417.823,Z 950.811,A -85,B 0,C 180,E1 15902.16,E2 15902.16} C_VEL
LIN {X 0,Y 438.59,Z 1009.27,A -85,B 0,C 180,E1 15904.637,E2 15904.637} C_VEL
LIN {X 0,Y 436.926,Z 1063.304,A -85,B 0,C 180,E1 15906.198,E2 15906.198} C_VEL
LIN {X 0,Y 432.468,Z 1108.675,A -85,B 0,C 180,E1 15909.543,E2 15909.543} C_VEL
LIN {X 0,Y 427.201,Z 1144.417,A -85,B 0,C 180,E1 15914.499,E2 15914.499} C_VEL
LIN {X 0,Y 423.07,Z 1168.02,A -85,B 0,C 180,E1 15920.73,E2 15920.73} C_VEL
LIN {X 0,Y 421.52,Z 1177.289,A -85,B 0,C 180,E1 15926.854,E2 15926.854} C_VEL
LIN {X 0,Y 421.601,Z 1175.188,A -85,B 0,C 180,E1 15933.044,E2 15933.044} C_VEL
LIN {X 0,Y 424.004,Z 1159.202,A -85,B 0,C 180,E1 15939.737,E2 15939.737} C_VEL
LIN {X 0,Y 428.454,Z 1130.764,A -85,B 0,C 180,E1 15945.35,E2 15945.35} C_VEL
LIN {X 0,Y 433.69,Z 1091.093,A -85,B 0,C 180,E1 15949.625,E2 15949.625} C_VEL
LIN {X 0,Y 436.992,Z 1042.711,A -85,B 0,C 180,E1 15952.237,E2 15952.237} C_VEL
LIN {X 0,Y 435.454,Z 1001.281,A -85,B 0,C 180,E1 15953.228,E2 15953.228} C_VEL
LIN {X 0,Y 417.509,Z 948.94,A -85,B 0,C 180,E1 15955.51,E2 15955.51} C_VEL
LIN {X 0,Y 417.035,Z 948.94,A -85,B 0,C 180,E1 15964.99,E2 15964.99} C_VEL
LIN {X 0,Y 417.156,Z 948.94,A -85,B 0,C 180,E1 15975.101,E2 15975.101} C_VEL
LIN {X 0,Y 417.275,Z 948.94,A -85,B 0,C 180,E1 15985.656,E2 15985.656} C_VEL
LIN {X 0,Y 417.64,Z 948.94,A -85,B 0,C 180,E1 15995.273,E2 15995.273} C_VEL
LIN {X 0,Y 418.557,Z 948.94,A -85,B 0,C 180,E1 16006.346,E2 16006.346} C_VEL
LIN {X 0,Y 418.987,Z 948.94,A -85,B 0,C 180,E1 16016.941,E2 16016.941} C_VEL
LIN {X 0,Y 418.501,Z 948.94,A -85,B 0,C 180,E1 16027.272,E2 16027.272} C_VEL
LIN {X 0,Y 417.745,Z 948.94,A -85,B 0,C 180,E1 16037.967,E2 16037.967} C_VEL
LIN {X 0,Y 417.537,Z 948.94,A -85,B 0,C 180,E1 16049.366,E2 16049.366} C_VEL
LIN {X 0,Y 417.705,Z 950.856,A -85,B 0,C 180,E1 16059.46,E2 16059.46} C_VEL
LIN {X 0,Y 454.37,Z 1030.073,A -85,B 0,C 180,E1 16066.953,E2 16066.953} C_VEL
LIN {X 0,Y 460.825,Z 1058.018,A -85,B 0,C 180,E1 16069.157,E2 16069.157} C_VEL
LIN {X 0,Y 445.666,Z 1131.668,A -85,B 0,C 180,E1 16074.113,E2 16074.113} C_VEL
LIN {X 0,Y 433.052,Z 1193.013,A -85,B 0,C 180,E1 16080.705,E2 16080.705} C_VEL
LIN {X 0,Y 424.549,Z 1240.409,A -85,B 0,C 180,E1 16088.566,E2 16088.566} C_VEL
LIN {X 0,Y 420.334,Z 1271.647,A -85,B 0,C 180,E1 16096.899,E2 16096.899} C_VEL
LIN {X 0,Y 419.549,Z 1287.094,A -85,B 0,C 180,E1 16104.864,E2 16104.864} C_VEL
LIN {X 0,Y 419.761,Z 1289.862,A -85,B 0,C 180,E1 16111.087,E2 16111.087} C_VEL
LIN {X 0,Y 419.651,Z 1281.221,A -85,B 0,C 180,E1 16118.891,E2 16118.891} C_VEL
LIN {X 0,Y 421.379,Z 1258.729,A -85,B 0,C 180,E1 16126.499,E2 16126.499} C_VEL
LIN {X 0,Y 426.332,Z 1220.106,A -85,B 0,C 180,E1 16133.935,E2 16133.935} C_VEL
LIN {X 0,Y 430.545,Z 1192.478,A -85,B 0,C 180,E1 16137.697,E2 16137.697} C_VEL
LIN {X 0,Y 427.565,Z 1168.002,A -85,B 0,C 180,E1 16141.103,E2 16141.103} C_VEL
LIN {X 0,Y 447.199,Z 1079.331,A -85,B 0,C 180,E1 16148.94,E2 16148.94} C_VEL
LIN {X 0,Y 456.224,Z 1045.933,A -85,B 0,C 180,E1 16151.469,E2 16151.469} C_VEL
LIN {X 0,Y 463.107,Z 1028.16,A -85,B 0,C 180,E1 16153.722,E2 16153.722} C_VEL
LIN {X 0,Y 459.691,Z 1065.832,A -85,B 0,C 180,E1 16156.718,E2 16156.718} C_VEL
LIN {X 0,Y 446.271,Z 1123.725,A -85,B 0,C 180,E1 16161.23,E2 16161.23} C_VEL
LIN {X 0,Y 432.152,Z 1171.042,A -85,B 0,C 180,E1 16167.432,E2 16167.432} C_VEL
LIN {X 0,Y 420.255,Z 1208.079,A -85,B 0,C 180,E1 16175.482,E2 16175.482} C_VEL
LIN {X 0,Y 413.789,Z 1230.386,A -85,B 0,C 180,E1 16184.053,E2 16184.053} C_VEL
LIN {X 0,Y 411.643,Z 1240.067,A -85,B 0,C 180,E1 16192.606,E2 16192.606} C_VEL
LIN {X 0,Y 411.624,Z 1238.27,A -85,B 0,C 180,E1 16201.077,E2 16201.077} C_VEL
LIN {X 0,Y 413.085,Z 1224.91,A -85,B 0,C 180,E1 16209.538,E2 16209.538} C_VEL
LIN {X 0,Y 418.658,Z 1195.82,A -85,B 0,C 180,E1 16218.517,E2 16218.517} C_VEL
LIN {X 0,Y 428.324,Z 1153.007,A -85,B 0,C 180,E1 16226.314,E2 16226.314} C_VEL
LIN {X 0,Y 440.085,Z 1098.39,A -85,B 0,C 180,E1 16232.485,E2 16232.485} C_VEL
LIN {X 0,Y 447.56,Z 1046.874,A -85,B 0,C 180,E1 16236.269,E2 16236.269} C_VEL
LIN {X 0,Y 425.3,Z 985.854,A -85,B 0,C 180,E1 16241.294,E2 16241.294} C_VEL
LIN {X 0,Y 409.059,Z 948.94,A -85,B 0,C 180,E1 16244.418,E2 16244.418} C_VEL
LIN {X 0,Y 409.191,Z 948.94,A -85,B 0,C 180,E1 16254.855,E2 16254.855} C_VEL
LIN {X 0,Y 409.715,Z 950.737,A -85,B 0,C 180,E1 16261.554,E2 16261.554} C_VEL
LIN {X 0,Y 431.415,Z 1012.269,A -85,B 0,C 180,E1 16264.236,E2 16264.236} C_VEL
LIN {X 0,Y 429.546,Z 1065.538,A -85,B 0,C 180,E1 16265.846,E2 16265.846} C_VEL
LIN {X 0,Y 424.876,Z 1110.732,A -85,B 0,C 180,E1 16269.297,E2 16269.297} C_VEL
LIN {X 0,Y 419.293,Z 1146.627,A -85,B 0,C 180,E1 16274.469,E2 16274.469} C_VEL
LIN {X 0,Y 415.262,Z 1168.774,A -85,B 0,C 180,E1 16280.484,E2 16280.484} C_VEL
LIN {X 0,Y 413.583,Z 1178.237,A -85,B 0,C 180,E1 16286.794,E2 16286.794} C_VEL
LIN {X 0,Y 413.671,Z 1176.153,A -85,B 0,C 180,E1 16293.102,E2 16293.102} C_VEL
LIN {X 0,Y 416.215,Z 1160.092,A -85,B 0,C 180,E1 16299.949,E2 16299.949} C_VEL
LIN {X 0,Y 421.082,Z 1130.047,A -85,B 0,C 180,E1 16305.894,E2 16305.894} C_VEL
LIN {X 0,Y 426.49,Z 1088.905,A -85,B 0,C 180,E1 16310.242,E2 16310.242} C_VEL
LIN {X 0,Y 429.798,Z 1041.322,A -85,B 0,C 180,E1 16312.72,E2 16312.72} C_VEL
LIN {X 0,Y 427.918,Z 1001.683,A -85,B 0,C 180,E1 16313.683,E2 16313.683} C_VEL
LIN {X 0,Y 409.449,Z 948.94,A -85,B 0,C 180,E1 16316.013,E2 16316.013} C_VEL
LIN {X 0,Y 408.988,Z 948.94,A -85,B 0,C 180,E1 16327.677,E2 16327.677} C_VEL
LIN {X 0,Y 409.077,Z 948.94,A -85,B 0,C 180,E1 16336.625,E2 16336.625} C_VEL
LIN {X 0,Y 409.288,Z 948.94,A -85,B 0,C 180,E1 16347.447,E2 16347.447} C_VEL
LIN {X 0,Y 409.644,Z 948.94,A -85,B 0,C 180,E1 16357.082,E2 16357.082} C_VEL
LIN {X 0,Y 410.65,Z 948.94,A -85,B 0,C 180,E1 16368.25,E2 16368.25} C_VEL
LIN {X 0,Y 410.788,Z 948.94,A -85,B 0,C 180,E1 16378.921,E2 16378.921} C_VEL
LIN {X 0,Y 410.463,Z 948.94,A -85,B 0,C 180,E1 16387.415,E2 16387.415} C_VEL
LIN {X 0,Y 409.684,Z 948.94,A -85,B 0,C 180,E1 16398.333,E2 16398.333} C_VEL
LIN {X 0,Y 409.527,Z 948.94,A -85,B 0,C 180,E1 16409.571,E2 16409.571} C_VEL
LIN {X 0,Y 409.675,Z 950.71,A -85,B 0,C 180,E1 16418.515,E2 16418.515} C_VEL
LIN {X 0,Y 447.07,Z 1031.978,A -85,B 0,C 180,E1 16426.463,E2 16426.463} C_VEL
LIN {X 0,Y 453.575,Z 1060.126,A -85,B 0,C 180,E1 16428.758,E2 16428.758} C_VEL
LIN {X 0,Y 437.72,Z 1134.662,A -85,B 0,C 180,E1 16433.955,E2 16433.955} C_VEL
LIN {X 0,Y 424.596,Z 1196.657,A -85,B 0,C 180,E1 16440.922,E2 16440.922} C_VEL
LIN {X 0,Y 416.141,Z 1242.773,A -85,B 0,C 180,E1 16448.947,E2 16448.947} C_VEL
LIN {X 0,Y 412.262,Z 1272.325,A -85,B 0,C 180,E1 16457.233,E2 16457.233} C_VEL
LIN {X 0,Y 411.572,Z 1286.452,A -85,B 0,C 180,E1 16464.764,E2 16464.764} C_VEL
LIN {X 0,Y 411.787,Z 1289.364,A -85,B 0,C 180,E1 16471.108,E2 16471.108} C_VEL
LIN {X 0,Y 411.68,Z 1280.796,A -85,B 0,C 180,E1 16479.064,E2 16479.064} C_VEL
LIN {X 0,Y 413.397,Z 1259.545,A -85,B 0,C 180,E1 16486.514,E2 16486.514} C_VEL
LIN {X 0,Y 418.589,Z 1221.615,A -85,B 0,C 180,E1 16494.122,E2 16494.122} C_VEL
LIN {X 0,Y 427.565,Z 1168.002,A -85,B 0,C 180,E1 16501.103,E2 16501.103} C_VEL
LIN {X 0,Y 426.618,Z 1142.794,A -85,B 0,C 180,E1 16504.459,E2 16504.459} C_VEL
LIN {X 0,Y 450.142,Z 1061.807,A -85,B 0,C 180,E1 16511.156,E2 16511.156} C_VEL
LIN {X 0,Y 459.48,Z 1038.573,A -85,B 0,C 180,E1 16513.533,E2 16513.533} C_VEL
LIN {X 0,Y 454.428,Z 1071.791,A -85,B 0,C 180,E1 16516.16,E2 16516.16} C_VEL
LIN {X 0,Y 439.721,Z 1128.571,A -85,B 0,C 180,E1 16520.863,E2 16520.863} C_VEL
LIN {X 0,Y 424.291,Z 1176.162,A -85,B 0,C 180,E1 16527.467,E2 16527.467} C_VEL
LIN {X 0,Y 412.298,Z 1210.923,A -85,B 0,C 180,E1 16535.557,E2 16535.557} C_VEL
LIN {X 0,Y 405.541,Z 1233.009,A -85,B 0,C 180,E1 16544.834,E2 16544.834} C_VEL
LIN {X 0,Y 403.679,Z 1240.666,A -85,B 0,C 180,E1 16552.459,E2 16552.459} C_VEL
LIN {X 0,Y 403.636,Z 1238.716,A -85,B 0,C 180,E1 16561.098,E2 16561.098} C_VEL
LIN {X 0,Y 405.172,Z 1225.147,A -85,B 0,C 180,E1 16569.726,E2 16569.726} C_VEL
LIN {X 0,Y 410.869,Z 1196.236,A -85,B 0,C 180,E1 16578.768,E2 16578.768} C_VEL
LIN {X 0,Y 420.586,Z 1154.4,A -85,B 0,C 180,E1 16586.548,E2 16586.548} C_VEL
LIN {X 0,Y 432.588,Z 1100.274,A -85,B 0,C 180,E1 16592.813,E2 16592.813} C_VEL
LIN {X 0,Y 440.531,Z 1049.719,A -85,B 0,C 180,E1 16596.611,E2 16596.611} C_VEL
LIN {X 0,Y 418.359,Z 988.395,A -85,B 0,C 180,E1 16601.811,E2 16601.811} C_VEL
LIN {X 0,Y 401.034,Z 948.94,A -85,B 0,C 180,E1 16605.023,E2 16605.023} C_VEL
LIN {X 0,Y 401.199,Z 948.94,A -85,B 0,C 180,E1 16616.681,E2 16616.681} C_VEL
LIN {X 0,Y 401.668,Z 950.856,A -85,B 0,C 180,E1 16620.929,E2 16620.929} C_VEL
LIN {X 0,Y 424.221,Z 1014.082,A -85,B 0,C 180,E1 16623.797,E2 16623.797} C_VEL
LIN {X 0,Y 422.184,Z 1067.388,A -85,B 0,C 180,E1 16625.465,E2 16625.465} C_VEL
LIN {X 0,Y 417.286,Z 1112.79,A -85,B 0,C 180,E1 16629.042,E2 16629.042} C_VEL
LIN {X 0,Y 411.632,Z 1147.521,A -85,B 0,C 180,E1 16634.172,E2 16634.172} C_VEL
LIN {X 0,Y 407.21,Z 1170.81,A -85,B 0,C 180,E1 16640.762,E2 16640.762} C_VEL
LIN {X 0,Y 405.664,Z 1179.182,A -85,B 0,C 180,E1 16646.731,E2 16646.731} C_VEL
LIN {X 0,Y 405.757,Z 1177.116,A -85,B 0,C 180,E1 16653.162,E2 16653.162} C_VEL
LIN {X 0,Y 408.392,Z 1161.191,A -85,B 0,C 180,E1 16660.111,E2 16660.111} C_VEL
LIN {X 0,Y 413.193,Z 1132.806,A -85,B 0,C 180,E1 16665.932,E2 16665.932} C_VEL
LIN {X 0,Y 418.816,Z 1093.254,A -85,B 0,C 180,E1 16670.353,E2 16670.353} C_VEL
LIN {X 0,Y 422.397,Z 1045.013,A -85,B 0,C 180,E1 16673.054,E2 16673.054} C_VEL
LIN {X 0,Y 420.755,Z 1003.523,A -85,B 0,C 180,E1 16674.106,E2 16674.106} C_VEL
LIN {X 0,Y 401.4,Z 948.94,A -85,B 0,C 180,E1 16676.609,E2 16676.609} C_VEL
LIN {X 0,Y 400.982,Z 948.94,A -85,B 0,C 180,E1 16685.843,E2 16685.843} C_VEL
LIN {X 0,Y 401.012,Z 948.94,A -85,B 0,C 180,E1 16697.465,E2 16697.465} C_VEL
LIN {X 0,Y 401.27,Z 948.94,A -85,B 0,C 180,E1 16708.193,E2 16708.193} C_VEL
LIN {X 0,Y 401.702,Z 948.94,A -85,B 0,C 180,E1 16718.942,E2 16718.942} C_VEL
LIN {X 0,Y 402.629,Z 948.94,A -85,B 0,C 180,E1 16728.012,E2 16728.012} C_VEL
LIN {X 0,Y 402.788,Z 948.94,A -85,B 0,C 180,E1 16738.899,E2 16738.899} C_VEL
LIN {X 0,Y 402.441,Z 948.94,A -85,B 0,C 180,E1 16747.564,E2 16747.564} C_VEL
LIN {X 0,Y 401.642,Z 948.94,A -85,B 0,C 180,E1 16758.714,E2 16758.714} C_VEL
LIN {X 0,Y 401.433,Z 948.94,A -85,B 0,C 180,E1 16768.18,E2 16768.18} C_VEL
LIN {X 0,Y 401.686,Z 950.88,A -85,B 0,C 180,E1 16777.554,E2 16777.554} C_VEL
LIN {X 0,Y 438.058,Z 1030.056,A -85,B 0,C 180,E1 16785.582,E2 16785.582} C_VEL
LIN {X 0,Y 446.255,Z 1062.014,A -85,B 0,C 180,E1 16788.346,E2 16788.346} C_VEL
LIN {X 0,Y 430.324,Z 1134.771,A -85,B 0,C 180,E1 16793.55,E2 16793.55} C_VEL
LIN {X 0,Y 416.874,Z 1196.575,A -85,B 0,C 180,E1 16800.63,E2 16800.63} C_VEL
LIN {X 0,Y 408.05,Z 1243.369,A -85,B 0,C 180,E1 16808.979,E2 16808.979} C_VEL
LIN {X 0,Y 404.236,Z 1272.843,A -85,B 0,C 180,E1 16817.559,E2 16817.559} C_VEL
LIN {X 0,Y 403.565,Z 1286.192,A -85,B 0,C 180,E1 16825.066,E2 16825.066} C_VEL
LIN {X 0,Y 403.5,Z 1287.915,A -85,B 0,C 180,E1 16833.287,E2 16833.287} C_VEL
LIN {X 0,Y 404.117,Z 1275.741,A -85,B 0,C 180,E1 16841.422,E2 16841.422} C_VEL
LIN {X 0,Y 407.427,Z 1247.675,A -85,B 0,C 180,E1 16849.638,E2 16849.638} C_VEL
LIN {X 0,Y 414.606,Z 1202.177,A -85,B 0,C 180,E1 16857.517,E2 16857.517} C_VEL
LIN {X 0,Y 426.618,Z 1142.794,A -85,B 0,C 180,E1 16864.459,E2 16864.459} C_VEL
LIN {X 0,Y 428.546,Z 1117.688,A -85,B 0,C 180,E1 16867.808,E2 16867.808} C_VEL
LIN {X 0,Y 453.232,Z 1054.593,A -85,B 0,C 180,E1 16873.126,E2 16873.126} C_VEL
LIN {X 0,Y 454.92,Z 1052.42,A -85,B 0,C 180,E1 16873.676,E2 16873.676} C_VEL
LIN {X 0,Y 436.193,Z 1124.172,A -85,B 0,C 180,E1 16879.464,E2 16879.464} C_VEL
LIN {X 0,Y 419.684,Z 1172.371,A -85,B 0,C 180,E1 16885.93,E2 16885.93} C_VEL
LIN {X 0,Y 406.016,Z 1209.286,A -85,B 0,C 180,E1 16894.248,E2 16894.248} C_VEL
LIN {X 0,Y 398.264,Z 1232.007,A -85,B 0,C 180,E1 16903.414,E2 16903.414} C_VEL
LIN {X 0,Y 395.742,Z 1241.273,A -85,B 0,C 180,E1 16912.307,E2 16912.307} C_VEL
LIN {X 0,Y 395.671,Z 1239.158,A -85,B 0,C 180,E1 16921.121,E2 16921.121} C_VEL
LIN {X 0,Y 397.263,Z 1225.365,A -85,B 0,C 180,E1 16929.922,E2 16929.922} C_VEL
LIN {X 0,Y 403.172,Z 1196.378,A -85,B 0,C 180,E1 16939.084,E2 16939.084} C_VEL
LIN {X 0,Y 413.282,Z 1153.871,A -85,B 0,C 180,E1 16947.055,E2 16947.055} C_VEL
LIN {X 0,Y 425.435,Z 1100.537,A -85,B 0,C 180,E1 16953.283,E2 16953.283} C_VEL
LIN {X 0,Y 433.143,Z 1051.366,A -85,B 0,C 180,E1 16957.065,E2 16957.065} C_VEL
LIN {X 0,Y 411.277,Z 990.401,A -85,B 0,C 180,E1 16962.376,E2 16962.376} C_VEL
LIN {X 0,Y 392.95,Z 948.94,A -85,B 0,C 180,E1 16966.125,E2 16966.125} C_VEL
LIN {X 0,Y 393.139,Z 948.94,A -85,B 0,C 180,E1 16976.143,E2 16976.143} C_VEL
LIN {X 0,Y 393.508,Z 950.417,A -85,B 0,C 180,E1 16980.253,E2 16980.253} C_VEL
LIN {X 0,Y 416.913,Z 1013.738,A -85,B 0,C 180,E1 16983.292,E2 16983.292} C_VEL
LIN {X 0,Y 415.064,Z 1067.143,A -85,B 0,C 180,E1 16984.957,E2 16984.957} C_VEL
LIN {X 0,Y 410.02,Z 1112.404,A -85,B 0,C 180,E1 16988.51,E2 16988.51} C_VEL
LIN {X 0,Y 404.002,Z 1148.412,A -85,B 0,C 180,E1 16993.865,E2 16993.865} C_VEL
LIN {X 0,Y 399.585,Z 1170.622,A -85,B 0,C 180,E1 17000.107,E2 17000.107} C_VEL
LIN {X 0,Y 397.728,Z 1180.13,A -85,B 0,C 180,E1 17006.666,E2 17006.666} C_VEL
LIN {X 0,Y 397.828,Z 1178.082,A -85,B 0,C 180,E1 17013.226,E2 17013.226} C_VEL
LIN {X 0,Y 400.587,Z 1162.182,A -85,B 0,C 180,E1 17020.31,E2 17020.31} C_VEL
LIN {X 0,Y 405.58,Z 1133.826,A -85,B 0,C 180,E1 17026.239,E2 17026.239} C_VEL
LIN {X 0,Y 411.407,Z 1094.334,A -85,B 0,C 180,E1 17030.736,E2 17030.736} C_VEL
LIN {X 0,Y 415.102,Z 1046.847,A -85,B 0,C 180,E1 17033.46,E2 17033.46} C_VEL
LIN {X 0,Y 413.44,Z 1004.735,A -85,B 0,C 180,E1 17034.566,E2 17034.566} C_VEL
LIN {X 0,Y 393.298,Z 948.94,A -85,B 0,C 180,E1 17037.441,E2 17037.441} C_VEL
LIN {X 0,Y 392.825,Z 948.94,A -85,B 0,C 180,E1 17047.584,E2 17047.584} C_VEL
LIN {X 0,Y 392.988,Z 948.94,A -85,B 0,C 180,E1 17058.756,E2 17058.756} C_VEL
LIN {X 0,Y 393.29,Z 948.94,A -85,B 0,C 180,E1 17070.12,E2 17070.12} C_VEL
LIN {X 0,Y 393.829,Z 948.94,A -85,B 0,C 180,E1 17080.855,E2 17080.855} C_VEL
LIN {X 0,Y 394.501,Z 948.94,A -85,B 0,C 180,E1 17090.008,E2 17090.008} C_VEL
LIN {X 0,Y 394.804,Z 948.94,A -85,B 0,C 180,E1 17098.877,E2 17098.877} C_VEL
LIN {X 0,Y 394.402,Z 948.94,A -85,B 0,C 180,E1 17107.719,E2 17107.719} C_VEL
LIN {X 0,Y 393.573,Z 948.94,A -85,B 0,C 180,E1 17119.343,E2 17119.343} C_VEL
LIN {X 0,Y 393.337,Z 948.94,A -85,B 0,C 180,E1 17129.892,E2 17129.892} C_VEL
LIN {X 0,Y 393.7,Z 950.914,A -85,B 0,C 180,E1 17136.557,E2 17136.557} C_VEL
LIN {X 0,Y 429.49,Z 1029.095,A -85,B 0,C 180,E1 17144.768,E2 17144.768} C_VEL
LIN {X 0,Y 439.131,Z 1062.975,A -85,B 0,C 180,E1 17147.872,E2 17147.872} C_VEL
LIN {X 0,Y 422.651,Z 1136.123,A -85,B 0,C 180,E1 17153.261,E2 17153.261} C_VEL
LIN {X 0,Y 408.97,Z 1197.46,A -85,B 0,C 180,E1 17160.478,E2 17160.478} C_VEL
LIN {X 0,Y 400.03,Z 1243.612,A -85,B 0,C 180,E1 17168.937,E2 17168.937} C_VEL
LIN {X 0,Y 396.263,Z 1272.396,A -85,B 0,C 180,E1 17177.514,E2 17177.514} C_VEL
LIN {X 0,Y 395.602,Z 1285.073,A -85,B 0,C 180,E1 17184.552,E2 17184.552} C_VEL
LIN {X 0,Y 395.797,Z 1288.308,A -85,B 0,C 180,E1 17191.152,E2 17191.152} C_VEL
LIN {X 0,Y 395.715,Z 1280.044,A -85,B 0,C 180,E1 17199.433,E2 17199.433} C_VEL
LIN {X 0,Y 398.063,Z 1257.547,A -85,B 0,C 180,E1 17207.578,E2 17207.578} C_VEL
LIN {X 0,Y 404.425,Z 1218.51,A -85,B 0,C 180,E1 17215.618,E2 17215.618} C_VEL
LIN {X 0,Y 418.561,Z 1152.995,A -85,B 0,C 180,E1 17224.247,E2 17224.247} C_VEL
LIN {X 0,Y 428.546,Z 1117.688,A -85,B 0,C 180,E1 17227.808,E2 17227.808} C_VEL
LIN {X 0,Y 435.435,Z 1093.478,A -85,B 0,C 180,E1 17231.122,E2 17231.122} C_VEL
LIN {X 0,Y 450.326,Z 1063.806,A -85,B 0,C 180,E1 17233.588,E2 17233.588} C_VEL
LIN {X 0,Y 430.122,Z 1128.943,A -85,B 0,C 180,E1 17238.983,E2 17238.983} C_VEL
LIN {X 0,Y 411.917,Z 1177.667,A -85,B 0,C 180,E1 17245.932,E2 17245.932} C_VEL
LIN {X 0,Y 397.695,Z 1213.204,A -85,B 0,C 180,E1 17254.597,E2 17254.597} C_VEL
LIN {X 0,Y 389.947,Z 1234.616,A -85,B 0,C 180,E1 17264.212,E2 17264.212} C_VEL
LIN {X 0,Y 387.782,Z 1241.891,A -85,B 0,C 180,E1 17272.148,E2 17272.148} C_VEL
LIN {X 0,Y 387.684,Z 1239.596,A -85,B 0,C 180,E1 17281.144,E2 17281.144} C_VEL
LIN {X 0,Y 389.36,Z 1225.558,A -85,B 0,C 180,E1 17290.125,E2 17290.125} C_VEL
LIN {X 0,Y 395.373,Z 1196.83,A -85,B 0,C 180,E1 17299.332,E2 17299.332} C_VEL
LIN {X 0,Y 405.571,Z 1155.144,A -85,B 0,C 180,E1 17307.31,E2 17307.31} C_VEL
LIN {X 0,Y 418.295,Z 1100.756,A -85,B 0,C 180,E1 17313.768,E2 17313.768} C_VEL
LIN {X 0,Y 425.906,Z 1053.675,A -85,B 0,C 180,E1 17317.467,E2 17317.467} C_VEL
LIN {X 0,Y 404.395,Z 993.11,A -85,B 0,C 180,E1 17322.899,E2 17322.899} C_VEL
LIN {X 0,Y 384.891,Z 948.94,A -85,B 0,C 180,E1 17326.88,E2 17326.88} C_VEL
LIN {X 0,Y 385.172,Z 948.94,A -85,B 0,C 180,E1 17337.953,E2 17337.953} C_VEL
LIN {X 0,Y 385.469,Z 950.615,A -85,B 0,C 180,E1 17339.568,E2 17339.568} C_VEL
LIN {X 0,Y 409.834,Z 1015.586,A -85,B 0,C 180,E1 17342.826,E2 17342.826} C_VEL
LIN {X 0,Y 407.749,Z 1068.918,A -85,B 0,C 180,E1 17344.541,E2 17344.541} C_VEL
LIN {X 0,Y 402.444,Z 1114.659,A -85,B 0,C 180,E1 17348.254,E2 17348.254} C_VEL
LIN {X 0,Y 396.373,Z 1149.305,A -85,B 0,C 180,E1 17353.546,E2 17353.546} C_VEL
LIN {X 0,Y 391.751,Z 1171.546,A -85,B 0,C 180,E1 17359.907,E2 17359.907} C_VEL
LIN {X 0,Y 389.81,Z 1181.076,A -85,B 0,C 180,E1 17366.598,E2 17366.598} C_VEL
LIN {X 0,Y 389.915,Z 1179.045,A -85,B 0,C 180,E1 17373.291,E2 17373.291} C_VEL
LIN {X 0,Y 392.794,Z 1163.173,A -85,B 0,C 180,E1 17380.517,E2 17380.517} C_VEL
LIN {X 0,Y 398.246,Z 1133.248,A -85,B 0,C 180,E1 17386.813,E2 17386.813} C_VEL
LIN {X 0,Y 404.292,Z 1092.143,A -85,B 0,C 180,E1 17391.406,E2 17391.406} C_VEL
LIN {X 0,Y 407.994,Z 1044.861,A -85,B 0,C 180,E1 17394.019,E2 17394.019} C_VEL
LIN {X 0,Y 406.13,Z 1005.978,A -85,B 0,C 180,E1 17395.044,E2 17395.044} C_VEL
LIN {X 0,Y 385.23,Z 948.94,A -85,B 0,C 180,E1 17397.99,E2 17397.99} C_VEL
LIN {X 0,Y 384.868,Z 948.94,A -85,B 0,C 180,E1 17409.699,E2 17409.699} C_VEL
LIN {X 0,Y 384.987,Z 948.94,A -85,B 0,C 180,E1 17420.133,E2 17420.133} C_VEL
LIN {X 0,Y 385.301,Z 948.94,A -85,B 0,C 180,E1 17430.476,E2 17430.476} C_VEL
LIN {X 0,Y 385.789,Z 948.94,A -85,B 0,C 180,E1 17440.44,E2 17440.44} C_VEL
LIN {X 0,Y 386.494,Z 948.94,A -85,B 0,C 180,E1 17449.799,E2 17449.799} C_VEL
LIN {X 0,Y 386.807,Z 948.94,A -85,B 0,C 180,E1 17458.854,E2 17458.854} C_VEL
LIN {X 0,Y 386.362,Z 948.94,A -85,B 0,C 180,E1 17467.881,E2 17467.881} C_VEL
LIN {X 0,Y 385.558,Z 948.94,A -85,B 0,C 180,E1 17479.526,E2 17479.526} C_VEL
LIN {X 0,Y 385.359,Z 948.94,A -85,B 0,C 180,E1 17489.469,E2 17489.469} C_VEL
LIN {X 0,Y 385.553,Z 950.425,A -85,B 0,C 180,E1 17495.486,E2 17495.486} C_VEL
LIN {X 0,Y 420.913,Z 1028.075,A -85,B 0,C 180,E1 17503.932,E2 17503.932} C_VEL
LIN {X 0,Y 431.972,Z 1064.286,A -85,B 0,C 180,E1 17507.416,E2 17507.416} C_VEL
LIN {X 0,Y 415.009,Z 1137.421,A -85,B 0,C 180,E1 17512.963,E2 17512.963} C_VEL
LIN {X 0,Y 401.049,Z 1198.308,A -85,B 0,C 180,E1 17520.318,E2 17520.318} C_VEL
LIN {X 0,Y 391.895,Z 1244.582,A -85,B 0,C 180,E1 17529.074,E2 17529.074} C_VEL
LIN {X 0,Y 388.242,Z 1272.353,A -85,B 0,C 180,E1 17537.644,E2 17537.644} C_VEL
LIN {X 0,Y 387.642,Z 1284.352,A -85,B 0,C 180,E1 17544.44,E2 17544.44} C_VEL
LIN {X 0,Y 387.802,Z 1287.767,A -85,B 0,C 180,E1 17551.176,E2 17551.176} C_VEL
LIN {X 0,Y 387.744,Z 1279.681,A -85,B 0,C 180,E1 17559.629,E2 17559.629} C_VEL
LIN {X 0,Y 390.288,Z 1257.652,A -85,B 0,C 180,E1 17567.867,E2 17567.867} C_VEL
LIN {X 0,Y 397.487,Z 1217.515,A -85,B 0,C 180,E1 17576.372,E2 17576.372} C_VEL
LIN {X 0,Y 414.443,Z 1148.956,A -85,B 0,C 180,E1 17585.623,E2 17585.623} C_VEL
LIN {X 0,Y 435.435,Z 1093.478,A -85,B 0,C 180,E1 17591.122,E2 17591.122} C_VEL
LIN {X 0,Y 443.368,Z 1079.154,A -85,B 0,C 180,E1 17593.41,E2 17593.41} C_VEL
LIN {X 0,Y 420.606,Z 1142.939,A -85,B 0,C 180,E1 17599.624,E2 17599.624} C_VEL
LIN {X 0,Y 401.621,Z 1188.484,A -85,B 0,C 180,E1 17607.119,E2 17607.119} C_VEL
LIN {X 0,Y 387.929,Z 1220.43,A -85,B 0,C 180,E1 17616.251,E2 17616.251} C_VEL
LIN {X 0,Y 381.356,Z 1238.359,A -85,B 0,C 180,E1 17626.207,E2 17626.207} C_VEL
LIN {X 0,Y 379.541,Z 1242.953,A -85,B 0,C 180,E1 17634.285,E2 17634.285} C_VEL
LIN {X 0,Y 379.695,Z 1237.645,A -85,B 0,C 180,E1 17643.46,E2 17643.46} C_VEL
LIN {X 0,Y 382.915,Z 1218.575,A -85,B 0,C 180,E1 17653.211,E2 17653.211} C_VEL
LIN {X 0,Y 390.65,Z 1184.165,A -85,B 0,C 180,E1 17662.585,E2 17662.585} C_VEL
LIN {X 0,Y 402.851,Z 1136.776,A -85,B 0,C 180,E1 17670.331,E2 17670.331} C_VEL
LIN {X 0,Y 415.62,Z 1079.581,A -85,B 0,C 180,E1 17676.102,E2 17676.102} C_VEL
LIN {X 0,Y 418.195,Z 1054.491,A -85,B 0,C 180,E1 17678.025,E2 17678.025} C_VEL
LIN {X 0,Y 396.965,Z 994.301,A -85,B 0,C 180,E1 17683.551,E2 17683.551} C_VEL
LIN {X 0,Y 376.821,Z 948.94,A -85,B 0,C 180,E1 17687.657,E2 17687.657} C_VEL
LIN {X 0,Y 377.333,Z 950.35,A -85,B 0,C 180,E1 17698.83,E2 17698.83} C_VEL
LIN {X 0,Y 402.663,Z 1016.83,A -85,B 0,C 180,E1 17702.322,E2 17702.322} C_VEL
LIN {X 0,Y 400.707,Z 1068.742,A -85,B 0,C 180,E1 17704.006,E2 17704.006} C_VEL
LIN {X 0,Y 395.396,Z 1113.44,A -85,B 0,C 180,E1 17707.597,E2 17707.597} C_VEL
LIN {X 0,Y 388.96,Z 1149.294,A -85,B 0,C 180,E1 17713.023,E2 17713.023} C_VEL
LIN {X 0,Y 383.926,Z 1172.47,A -85,B 0,C 180,E1 17719.699,E2 17719.699} C_VEL
LIN {X 0,Y 381.89,Z 1182.022,A -85,B 0,C 180,E1 17726.527,E2 17726.527} C_VEL
LIN {X 0,Y 382.015,Z 1180.007,A -85,B 0,C 180,E1 17733.359,E2 17733.359} C_VEL
LIN {X 0,Y 384.996,Z 1164.165,A -85,B 0,C 180,E1 17740.733,E2 17740.733} C_VEL
LIN {X 0,Y 390.376,Z 1135.869,A -85,B 0,C 180,E1 17746.89,E2 17746.89} C_VEL
LIN {X 0,Y 396.635,Z 1096.495,A -85,B 0,C 180,E1 17751.546,E2 17751.546} C_VEL
LIN {X 0,Y 400.667,Z 1048.549,A -85,B 0,C 180,E1 17754.39,E2 17754.39} C_VEL
LIN {X 0,Y 399.072,Z 1008.046,A -85,B 0,C 180,E1 17755.507,E2 17755.507} C_VEL
LIN {X 0,Y 377.18,Z 948.94,A -85,B 0,C 180,E1 17758.625,E2 17758.625} C_VEL
LIN {X 0,Y 376.785,Z 948.94,A -85,B 0,C 180,E1 17768.548,E2 17768.548} C_VEL
LIN {X 0,Y 376.865,Z 948.94,A -85,B 0,C 180,E1 17778.324,E2 17778.324} C_VEL
LIN {X 0,Y 377.198,Z 948.94,A -85,B 0,C 180,E1 17789.776,E2 17789.776} C_VEL
LIN {X 0,Y 377.796,Z 948.94,A -85,B 0,C 180,E1 17800.526,E2 17800.526} C_VEL
LIN {X 0,Y 378.473,Z 948.94,A -85,B 0,C 180,E1 17809.58,E2 17809.58} C_VEL
LIN {X 0,Y 378.829,Z 948.94,A -85,B 0,C 180,E1 17818.83,E2 17818.83} C_VEL
LIN {X 0,Y 378.324,Z 948.94,A -85,B 0,C 180,E1 17828.049,E2 17828.049} C_VEL
LIN {X 0,Y 377.509,Z 948.94,A -85,B 0,C 180,E1 17839.959,E2 17839.959} C_VEL
LIN {X 0,Y 377.268,Z 948.94,A -85,B 0,C 180,E1 17850.268,E2 17850.268} C_VEL
LIN {X 0,Y 377.529,Z 950.717,A -85,B 0,C 180,E1 17854.428,E2 17854.428} C_VEL
LIN {X 0,Y 411.886,Z 1025.937,A -85,B 0,C 180,E1 17862.95,E2 17862.95} C_VEL
LIN {X 0,Y 424.935,Z 1065.033,A -85,B 0,C 180,E1 17866.914,E2 17866.914} C_VEL
LIN {X 0,Y 407.418,Z 1138.361,A -85,B 0,C 180,E1 17872.623,E2 17872.623} C_VEL
LIN {X 0,Y 393.272,Z 1198.362,A -85,B 0,C 180,E1 17880.048,E2 17880.048} C_VEL
LIN {X 0,Y 383.973,Z 1244.308,A -85,B 0,C 180,E1 17888.924,E2 17888.924} C_VEL
LIN {X 0,Y 380.241,Z 1272.442,A -85,B 0,C 180,E1 17897.843,E2 17897.843} C_VEL
LIN {X 0,Y 379.614,Z 1285.772,A -85,B 0,C 180,E1 17906.619,E2 17906.619} C_VEL
LIN {X 0,Y 379.543,Z 1286.491,A -85,B 0,C 180,E1 17913.494,E2 17913.494} C_VEL
LIN {X 0,Y 380.406,Z 1274.497,A -85,B 0,C 180,E1 17922.272,E2 17922.272} C_VEL
LIN {X 0,Y 384.613,Z 1246.36,A -85,B 0,C 180,E1 17931.158,E2 17931.158} C_VEL
LIN {X 0,Y 394.914,Z 1198.653,A -85,B 0,C 180,E1 17940.086,E2 17940.086} C_VEL
LIN {X 0,Y 422.592,Z 1118.346,A -85,B 0,C 180,E1 17949.991,E2 17949.991} C_VEL
LIN {X 0,Y 443.368,Z 1079.154,A -85,B 0,C 180,E1 17953.41,E2 17953.41} C_VEL
LIN {X 0,Y 440.083,Z 1088.551,A -85,B 0,C 180,E1 17954.102,E2 17954.102} C_VEL
LIN {X 0,Y 430.005,Z 1109.908,A -85,B 0,C 180,E1 17954.964,E2 17954.964} C_VEL
LIN {X 0,Y 408.198,Z 1161.983,A -85,B 0,C 180,E1 17961.241,E2 17961.241} C_VEL
LIN {X 0,Y 389.672,Z 1202.206,A -85,B 0,C 180,E1 17969.422,E2 17969.422} C_VEL
LIN {X 0,Y 377.432,Z 1229.572,A -85,B 0,C 180,E1 17979.422,E2 17979.422} C_VEL
LIN {X 0,Y 372.411,Z 1242.089,A -85,B 0,C 180,E1 17989.455,E2 17989.455} C_VEL
LIN {X 0,Y 371.728,Z 1242.173,A -85,B 0,C 180,E1 17998.853,E2 17998.853} C_VEL
LIN {X 0,Y 372.974,Z 1229.559,A -85,B 0,C 180,E1 18008.801,E2 18008.801} C_VEL
LIN {X 0,Y 377.974,Z 1204.035,A -85,B 0,C 180,E1 18018.156,E2 18018.156} C_VEL
LIN {X 0,Y 388.207,Z 1164.234,A -85,B 0,C 180,E1 18026.744,E2 18026.744} C_VEL
LIN {X 0,Y 401.416,Z 1112.29,A -85,B 0,C 180,E1 18033.664,E2 18033.664} C_VEL
LIN {X 0,Y 411.127,Z 1057.383,A -85,B 0,C 180,E1 18038.379,E2 18038.379} C_VEL
LIN {X 0,Y 390.374,Z 997.541,A -85,B 0,C 180,E1 18044.046,E2 18044.046} C_VEL
LIN {X 0,Y 368.775,Z 948.94,A -85,B 0,C 180,E1 18048.774,E2 18048.774} C_VEL
LIN {X 0,Y 369.308,Z 950.54,A -85,B 0,C 180,E1 18058.073,E2 18058.073} C_VEL
LIN {X 0,Y 395.47,Z 1018.248,A -85,B 0,C 180,E1 18061.799,E2 18061.799} C_VEL
LIN {X 0,Y 393.308,Z 1071.397,A -85,B 0,C 180,E1 18063.603,E2 18063.603} C_VEL
LIN {X 0,Y 387.551,Z 1117.12,A -85,B 0,C 180,E1 18067.47,E2 18067.47} C_VEL
LIN {X 0,Y 380.897,Z 1152.136,A -85,B 0,C 180,E1 18073.099,E2 18073.099} C_VEL
LIN {X 0,Y 375.824,Z 1174.68,A -85,B 0,C 180,E1 18080.062,E2 18080.062} C_VEL
LIN {X 0,Y 373.973,Z 1182.968,A -85,B 0,C 180,E1 18086.454,E2 18086.454} C_VEL
LIN {X 0,Y 374.103,Z 1180.971,A -85,B 0,C 180,E1 18093.43,E2 18093.43} C_VEL
LIN {X 0,Y 377.209,Z 1165.156,A -85,B 0,C 180,E1 18100.957,E2 18100.957} C_VEL
LIN {X 0,Y 382.79,Z 1136.89,A -85,B 0,C 180,E1 18107.235,E2 18107.235} C_VEL
LIN {X 0,Y 389.277,Z 1097.575,A -85,B 0,C 180,E1 18111.974,E2 18111.974} C_VEL
LIN {X 0,Y 393.416,Z 1050.71,A -85,B 0,C 180,E1 18114.831,E2 18114.831} C_VEL
LIN {X 0,Y 391.971,Z 1009.93,A -85,B 0,C 180,E1 18115.996,E2 18115.996} C_VEL
LIN {X 0,Y 369.109,Z 948.94,A -85,B 0,C 180,E1 18119.387,E2 18119.387} C_VEL
LIN {X 0,Y 368.659,Z 948.94,A -85,B 0,C 180,E1 18130.353,E2 18130.353} C_VEL
LIN {X 0,Y 368.812,Z 948.94,A -85,B 0,C 180,E1 18140.336,E2 18140.336} C_VEL
LIN {X 0,Y 369.237,Z 948.94,A -85,B 0,C 180,E1 18151.941,E2 18151.941} C_VEL
LIN {X 0,Y 369.87,Z 948.94,A -85,B 0,C 180,E1 18162.051,E2 18162.051} C_VEL
LIN {X 0,Y 370.398,Z 948.94,A -85,B 0,C 180,E1 18171.731,E2 18171.731} C_VEL
LIN {X 0,Y 370.655,Z 948.94,A -85,B 0,C 180,E1 18181.15,E2 18181.15} C_VEL
LIN {X 0,Y 370.11,Z 948.94,A -85,B 0,C 180,E1 18190.611,E2 18190.611} C_VEL
LIN {X 0,Y 369.424,Z 948.94,A -85,B 0,C 180,E1 18202.618,E2 18202.618} C_VEL
LIN {X 0,Y 369.493,Z 950.87,A -85,B 0,C 180,E1 18213.323,E2 18213.323} C_VEL
LIN {X 0,Y 402.955,Z 1023.949,A -85,B 0,C 180,E1 18221.951,E2 18221.951} C_VEL
LIN {X 0,Y 417.585,Z 1067.053,A -85,B 0,C 180,E1 18226.481,E2 18226.481} C_VEL
LIN {X 0,Y 399.136,Z 1142.045,A -85,B 0,C 180,E1 18232.553,E2 18232.553} C_VEL
LIN {X 0,Y 384.774,Z 1201.753,A -85,B 0,C 180,E1 18240.308,E2 18240.308} C_VEL
LIN {X 0,Y 375.593,Z 1246.294,A -85,B 0,C 180,E1 18249.361,E2 18249.361} C_VEL
LIN {X 0,Y 372.191,Z 1273.761,A -85,B 0,C 180,E1 18258.647,E2 18258.647} C_VEL
LIN {X 0,Y 371.64,Z 1285.105,A -85,B 0,C 180,E1 18266.547,E2 18266.547} C_VEL
LIN {X 0,Y 371.567,Z 1286.031,A -85,B 0,C 180,E1 18273.569,E2 18273.569} C_VEL
LIN {X 0,Y 372.399,Z 1274.852,A -85,B 0,C 180,E1 18282.276,E2 18282.276} C_VEL
LIN {X 0,Y 376.806,Z 1247.787,A -85,B 0,C 180,E1 18291.309,E2 18291.309} C_VEL
LIN {X 0,Y 388.138,Z 1200.248,A -85,B 0,C 180,E1 18300.667,E2 18300.667} C_VEL
LIN {X 0,Y 418.301,Z 1123.889,A -85,B 0,C 180,E1 18310.657,E2 18310.657} C_VEL
LIN {X 0,Y 436.073,Z 1094.181,A -85,B 0,C 180,E1 18313.482,E2 18313.482} C_VEL
LIN {X 0,Y 430.005,Z 1109.908,A -85,B 0,C 180,E1 18314.964,E2 18314.964} C_VEL
LIN {X 0,Y 414.699,Z 1138.642,A -85,B 0,C 180,E1 18316.861,E2 18316.861} C_VEL
LIN {X 0,Y 391.831,Z 1185.99,A -85,B 0,C 180,E1 18324.466,E2 18324.466} C_VEL
LIN {X 0,Y 375.307,Z 1218.847,A -85,B 0,C 180,E1 18333.636,E2 18333.636} C_VEL
LIN {X 0,Y 366.146,Z 1238.756,A -85,B 0,C 180,E1 18344.393,E2 18344.393} C_VEL
LIN {X 0,Y 363.612,Z 1244.125,A -85,B 0,C 180,E1 18354.033,E2 18354.033} C_VEL
LIN {X 0,Y 363.74,Z 1238.296,A -85,B 0,C 180,E1 18363.612,E2 18363.612} C_VEL
LIN {X 0,Y 367.186,Z 1218.813,A -85,B 0,C 180,E1 18373.747,E2 18373.747} C_VEL
LIN {X 0,Y 375.271,Z 1184.801,A -85,B 0,C 180,E1 18383.25,E2 18383.25} C_VEL
LIN {X 0,Y 388.121,Z 1137.277,A -85,B 0,C 180,E1 18391.237,E2 18391.237} C_VEL
LIN {X 0,Y 401.591,Z 1079.748,A -85,B 0,C 180,E1 18397.184,E2 18397.184} C_VEL
LIN {X 0,Y 403.831,Z 1059.442,A -85,B 0,C 180,E1 18398.817,E2 18398.817} C_VEL
LIN {X 0,Y 383.437,Z 1000.121,A -85,B 0,C 180,E1 18404.602,E2 18404.602} C_VEL
LIN {X 0,Y 360.783,Z 948.94,A -85,B 0,C 180,E1 18409.749,E2 18409.749} C_VEL
LIN {X 0,Y 361.166,Z 950.352,A -85,B 0,C 180,E1 18417.255,E2 18417.255} C_VEL
LIN {X 0,Y 388.206,Z 1019.067,A -85,B 0,C 180,E1 18421.236,E2 18421.236} C_VEL
LIN {X 0,Y 386.189,Z 1072.12,A -85,B 0,C 180,E1 18423.078,E2 18423.078} C_VEL
LIN {X 0,Y 380.255,Z 1117.817,A -85,B 0,C 180,E1 18426.996,E2 18426.996} C_VEL
LIN {X 0,Y 373.346,Z 1152.844,A -85,B 0,C 180,E1 18432.703,E2 18432.703} C_VEL
LIN {X 0,Y 367.987,Z 1175.605,A -85,B 0,C 180,E1 18439.849,E2 18439.849} C_VEL
LIN {X 0,Y 366.046,Z 1183.915,A -85,B 0,C 180,E1 18446.377,E2 18446.377} C_VEL
LIN {X 0,Y 366.198,Z 1181.933,A -85,B 0,C 180,E1 18453.505,E2 18453.505} C_VEL
LIN {X 0,Y 369.419,Z 1166.148,A -85,B 0,C 180,E1 18461.191,E2 18461.191} C_VEL
LIN {X 0,Y 375.507,Z 1136.508,A -85,B 0,C 180,E1 18467.832,E2 18467.832} C_VEL
LIN {X 0,Y 382.262,Z 1095.382,A -85,B 0,C 180,E1 18472.707,E2 18472.707} C_VEL
LIN {X 0,Y 386.414,Z 1048.694,A -85,B 0,C 180,E1 18475.449,E2 18475.449} C_VEL
LIN {X 0,Y 384.805,Z 1011.535,A -85,B 0,C 180,E1 18476.516,E2 18476.516} C_VEL
LIN {X 0,Y 361.047,Z 948.94,A -85,B 0,C 180,E1 18480.052,E2 18480.052} C_VEL
LIN {X 0,Y 360.663,Z 948.94,A -85,B 0,C 180,E1 18492.534,E2 18492.534} C_VEL
LIN {X 0,Y 360.786,Z 948.94,A -85,B 0,C 180,E1 18502.38,E2 18502.38} C_VEL
LIN {X 0,Y 361.374,Z 948.94,A -85,B 0,C 180,E1 18514.378,E2 18514.378} C_VEL
LIN {X 0,Y 362.359,Z 948.94,A -85,B 0,C 180,E1 18526.657,E2 18526.657} C_VEL
LIN {X 0,Y 362.834,Z 948.94,A -85,B 0,C 180,E1 18538.778,E2 18538.778} C_VEL
LIN {X 0,Y 362.272,Z 948.94,A -85,B 0,C 180,E1 18548.408,E2 18548.408} C_VEL
LIN {X 0,Y 361.433,Z 948.94,A -85,B 0,C 180,E1 18559.353,E2 18559.353} C_VEL
LIN {X 0,Y 361.212,Z 948.94,A -85,B 0,C 180,E1 18570.676,E2 18570.676} C_VEL
LIN {X 0,Y 361.512,Z 951.046,A -85,B 0,C 180,E1 18572.211,E2 18572.211} C_VEL
LIN {X 0,Y 393.926,Z 1021.796,A -85,B 0,C 180,E1 18580.892,E2 18580.892} C_VEL
LIN {X 0,Y 410.486,Z 1067.901,A -85,B 0,C 180,E1 18585.977,E2 18585.977} C_VEL
LIN {X 0,Y 391.715,Z 1142.206,A -85,B 0,C 180,E1 18592.126,E2 18592.126} C_VEL
LIN {X 0,Y 376.777,Z 1202.623,A -85,B 0,C 180,E1 18600.176,E2 18600.176} C_VEL
LIN {X 0,Y 367.419,Z 1247.084,A -85,B 0,C 180,E1 18609.513,E2 18609.513} C_VEL
LIN {X 0,Y 364.225,Z 1273.427,A -85,B 0,C 180,E1 18618.721,E2 18618.721} C_VEL
LIN {X 0,Y 363.657,Z 1284.415,A -85,B 0,C 180,E1 18626.471,E2 18626.471} C_VEL
LIN {X 0,Y 363.569,Z 1285.536,A -85,B 0,C 180,E1 18633.648,E2 18633.648} C_VEL
LIN {X 0,Y 364.451,Z 1274.864,A -85,B 0,C 180,E1 18642.421,E2 18642.421} C_VEL
LIN {X 0,Y 369.058,Z 1248.78,A -85,B 0,C 180,E1 18651.58,E2 18651.58} C_VEL
LIN {X 0,Y 381.904,Z 1200.786,A -85,B 0,C 180,E1 18661.491,E2 18661.491} C_VEL
LIN {X 0,Y 414.184,Z 1129.565,A -85,B 0,C 180,E1 18671.324,E2 18671.324} C_VEL
LIN {X 0,Y 427.845,Z 1108.976,A -85,B 0,C 180,E1 18673.47,E2 18673.47} C_VEL
LIN {X 0,Y 414.699,Z 1138.642,A -85,B 0,C 180,E1 18676.861,E2 18676.861} C_VEL
LIN {X 0,Y 398.437,Z 1164.649,A -85,B 0,C 180,E1 18679.369,E2 18679.369} C_VEL
LIN {X 0,Y 376.321,Z 1205.337,A -85,B 0,C 180,E1 18688.088,E2 18688.088} C_VEL
LIN {X 0,Y 362.309,Z 1231.816,A -85,B 0,C 180,E1 18698.536,E2 18698.536} C_VEL
LIN {X 0,Y 356.607,Z 1243.529,A -85,B 0,C 180,E1 18708.982,E2 18708.982} C_VEL
LIN {X 0,Y 355.743,Z 1243.112,A -85,B 0,C 180,E1 18718.802,E2 18718.802} C_VEL
LIN {X 0,Y 357.142,Z 1229.912,A -85,B 0,C 180,E1 18729.194,E2 18729.194} C_VEL
LIN {X 0,Y 362.911,Z 1202.731,A -85,B 0,C 180,E1 18739.214,E2 18739.214} C_VEL
LIN {X 0,Y 374.218,Z 1161.212,A -85,B 0,C 180,E1 18748.158,E2 18748.158} C_VEL
LIN {X 0,Y 388.341,Z 1107.513,A -85,B 0,C 180,E1 18755.231,E2 18755.231} C_VEL
LIN {X 0,Y 396.737,Z 1062.328,A -85,B 0,C 180,E1 18759.17,E2 18759.17} C_VEL
LIN {X 0,Y 377.012,Z 1003.85,A -85,B 0,C 180,E1 18765.057,E2 18765.057} C_VEL
LIN {X 0,Y 352.739,Z 948.94,A -85,B 0,C 180,E1 18770.724,E2 18770.724} C_VEL
LIN {X 0,Y 353.073,Z 950.29,A -85,B 0,C 180,E1 18776.4,E2 18776.4} C_VEL
LIN {X 0,Y 380.623,Z 1018.635,A -85,B 0,C 180,E1 18780.595,E2 18780.595} C_VEL
LIN {X 0,Y 379.349,Z 1071.03,A -85,B 0,C 180,E1 18782.435,E2 18782.435} C_VEL
LIN {X 0,Y 373.286,Z 1116.834,A -85,B 0,C 180,E1 18786.306,E2 18786.306} C_VEL
LIN {X 0,Y 366.041,Z 1152.664,A -85,B 0,C 180,E1 18792.086,E2 18792.086} C_VEL
LIN {X 0,Y 360.504,Z 1175.24,A -85,B 0,C 180,E1 18799.022,E2 18799.022} C_VEL
LIN {X 0,Y 358.129,Z 1184.861,A -85,B 0,C 180,E1 18806.296,E2 18806.296} C_VEL
LIN {X 0,Y 358.424,Z 1181.923,A -85,B 0,C 180,E1 18814.42,E2 18814.42} C_VEL
LIN {X 0,Y 362.35,Z 1164.258,A -85,B 0,C 180,E1 18822.331,E2 18822.331} C_VEL
LIN {X 0,Y 368.975,Z 1132.641,A -85,B 0,C 180,E1 18828.98,E2 18828.98} C_VEL
LIN {X 0,Y 375.564,Z 1091.334,A -85,B 0,C 180,E1 18833.608,E2 18833.608} C_VEL
LIN {X 0,Y 379.573,Z 1041.61,A -85,B 0,C 180,E1 18836.241,E2 18836.241} C_VEL
LIN {X 0,Y 377.573,Z 1012.691,A -85,B 0,C 180,E1 18837.073,E2 18837.073} C_VEL
LIN {X 0,Y 352.9,Z 948.94,A -85,B 0,C 180,E1 18841.077,E2 18841.077} C_VEL
LIN {X 0,Y 352.643,Z 948.94,A -85,B 0,C 180,E1 18851.746,E2 18851.746} C_VEL
LIN {X 0,Y 352.764,Z 948.94,A -85,B 0,C 180,E1 18862.621,E2 18862.621} C_VEL
LIN {X 0,Y 353.17,Z 948.94,A -85,B 0,C 180,E1 18873.149,E2 18873.149} C_VEL
LIN {X 0,Y 354.102,Z 948.94,A -85,B 0,C 180,E1 18884.371,E2 18884.371} C_VEL
LIN {X 0,Y 354.791,Z 948.94,A -85,B 0,C 180,E1 18896.73,E2 18896.73} C_VEL
LIN {X 0,Y 354.564,Z 948.94,A -85,B 0,C 180,E1 18906.119,E2 18906.119} C_VEL
LIN {X 0,Y 353.462,Z 948.94,A -85,B 0,C 180,E1 18918.762,E2 18918.762} C_VEL
LIN {X 0,Y 353.438,Z 950.779,A -85,B 0,C 180,E1 18931.017,E2 18931.017} C_VEL
LIN {X 0,Y 385.439,Z 1020.842,A -85,B 0,C 180,E1 18939.947,E2 18939.947} C_VEL
LIN {X 0,Y 403.028,Z 1070.146,A -85,B 0,C 180,E1 18945.565,E2 18945.565} C_VEL
LIN {X 0,Y 383.765,Z 1144.337,A -85,B 0,C 180,E1 18951.919,E2 18951.919} C_VEL
LIN {X 0,Y 368.549,Z 1204.267,A -85,B 0,C 180,E1 18960.189,E2 18960.189} C_VEL
LIN {X 0,Y 359.328,Z 1247.824,A -85,B 0,C 180,E1 18969.677,E2 18969.677} C_VEL
LIN {X 0,Y 356.216,Z 1273.498,A -85,B 0,C 180,E1 18979.011,E2 18979.011} C_VEL
LIN {X 0,Y 355.678,Z 1283.672,A -85,B 0,C 180,E1 18986.392,E2 18986.392} C_VEL
LIN {X 0,Y 355.577,Z 1285.029,A -85,B 0,C 180,E1 18993.73,E2 18993.73} C_VEL
LIN {X 0,Y 356.555,Z 1274.391,A -85,B 0,C 180,E1 19002.848,E2 19002.848} C_VEL
LIN {X 0,Y 361.699,Z 1247.953,A -85,B 0,C 180,E1 19012.396,E2 19012.396} C_VEL
LIN {X 0,Y 377.119,Z 1198.037,A -85,B 0,C 180,E1 19022.966,E2 19022.966} C_VEL
LIN {X 0,Y 411.137,Z 1133.927,A -85,B 0,C 180,E1 19032.161,E2 19032.161} C_VEL
LIN {X 0,Y 420.31,Z 1121.964,A -85,B 0,C 180,E1 19033.797,E2 19033.797} C_VEL
LIN {X 0,Y 398.437,Z 1164.649,A -85,B 0,C 180,E1 19039.369,E2 19039.369} C_VEL
LIN {X 0,Y 381.36,Z 1187.672,A -85,B 0,C 180,E1 19042.442,E2 19042.442} C_VEL
LIN {X 0,Y 361.49,Z 1221.171,A -85,B 0,C 180,E1 19052.277,E2 19052.277} C_VEL
LIN {X 0,Y 350.618,Z 1240.549,A -85,B 0,C 180,E1 19063.683,E2 19063.683} C_VEL
LIN {X 0,Y 347.679,Z 1245.322,A -85,B 0,C 180,E1 19073.759,E2 19073.759} C_VEL
LIN {X 0,Y 347.796,Z 1238.87,A -85,B 0,C 180,E1 19083.778,E2 19083.778} C_VEL
LIN {X 0,Y 351.201,Z 1220.278,A -85,B 0,C 180,E1 19093.776,E2 19093.776} C_VEL
LIN {X 0,Y 359.862,Z 1185.498,A -85,B 0,C 180,E1 19103.898,E2 19103.898} C_VEL
LIN {X 0,Y 373.249,Z 1138.26,A -85,B 0,C 180,E1 19112.112,E2 19112.112} C_VEL
LIN {X 0,Y 387.41,Z 1080.855,A -85,B 0,C 180,E1 19118.234,E2 19118.234} C_VEL
LIN {X 0,Y 389.071,Z 1063.107,A -85,B 0,C 180,E1 19119.761,E2 19119.761} C_VEL
LIN {X 0,Y 369.43,Z 1004.594,A -85,B 0,C 180,E1 19125.801,E2 19125.801} C_VEL
LIN {X 0,Y 344.685,Z 948.94,A -85,B 0,C 180,E1 19131.781,E2 19131.781} C_VEL
LIN {X 0,Y 344.988,Z 950.486,A -85,B 0,C 180,E1 19135.503,E2 19135.503} C_VEL
LIN {X 0,Y 372.927,Z 1017.958,A -85,B 0,C 180,E1 19139.907,E2 19139.907} C_VEL
LIN {X 0,Y 372.475,Z 1070.203,A -85,B 0,C 180,E1 19141.788,E2 19141.788} C_VEL
LIN {X 0,Y 366.571,Z 1115.015,A -85,B 0,C 180,E1 19145.493,E2 19145.493} C_VEL
LIN {X 0,Y 359.09,Z 1150.988,A -85,B 0,C 180,E1 19151.142,E2 19151.142} C_VEL
LIN {X 0,Y 353.014,Z 1174.797,A -85,B 0,C 180,E1 19158.158,E2 19158.158} C_VEL
LIN {X 0,Y 350.196,Z 1185.809,A -85,B 0,C 180,E1 19166.212,E2 19166.212} C_VEL
LIN {X 0,Y 350.508,Z 1182.892,A -85,B 0,C 180,E1 19174.52,E2 19174.52} C_VEL
LIN {X 0,Y 354.6,Z 1165.255,A -85,B 0,C 180,E1 19182.605,E2 19182.605} C_VEL
LIN {X 0,Y 361.131,Z 1135.11,A -85,B 0,C 180,E1 19189.162,E2 19189.162} C_VEL
LIN {X 0,Y 368.149,Z 1094.236,A -85,B 0,C 180,E1 19193.952,E2 19193.952} C_VEL
LIN {X 0,Y 372.366,Z 1046.219,A -85,B 0,C 180,E1 19196.67,E2 19196.67} C_VEL
LIN {X 0,Y 370.569,Z 1014.698,A -85,B 0,C 180,E1 19197.617,E2 19197.617} C_VEL
LIN {X 0,Y 344.801,Z 948.94,A -85,B 0,C 180,E1 19201.713,E2 19201.713} C_VEL
LIN {X 0,Y 344.554,Z 948.94,A -85,B 0,C 180,E1 19213.341,E2 19213.341} C_VEL
LIN {X 0,Y 344.838,Z 948.94,A -85,B 0,C 180,E1 19224.381,E2 19224.381} C_VEL
LIN {X 0,Y 345.249,Z 948.94,A -85,B 0,C 180,E1 19235.287,E2 19235.287} C_VEL
LIN {X 0,Y 346.225,Z 948.94,A -85,B 0,C 180,E1 19246.022,E2 19246.022} C_VEL
LIN {X 0,Y 346.831,Z 948.94,A -85,B 0,C 180,E1 19258.722,E2 19258.722} C_VEL
LIN {X 0,Y 346.045,Z 948.94,A -85,B 0,C 180,E1 19269.786,E2 19269.786} C_VEL
LIN {X 0,Y 345.291,Z 948.94,A -85,B 0,C 180,E1 19281.913,E2 19281.913} C_VEL
LIN {X 0,Y 345.359,Z 950.668,A -85,B 0,C 180,E1 19289.782,E2 19289.782} C_VEL
LIN {X 0,Y 376.897,Z 1019.772,A -85,B 0,C 180,E1 19298.951,E2 19298.951} C_VEL
LIN {X 0,Y 395.674,Z 1071.977,A -85,B 0,C 180,E1 19305.11,E2 19305.11} C_VEL
LIN {X 0,Y 376.024,Z 1145.661,A -85,B 0,C 180,E1 19311.615,E2 19311.615} C_VEL
LIN {X 0,Y 360.403,Z 1205.649,A -85,B 0,C 180,E1 19320.161,E2 19320.161} C_VEL
LIN {X 0,Y 351.225,Z 1248.483,A -85,B 0,C 180,E1 19329.847,E2 19329.847} C_VEL
LIN {X 0,Y 348.225,Z 1273.689,A -85,B 0,C 180,E1 19339.391,E2 19339.391} C_VEL
LIN {X 0,Y 347.619,Z 1284.432,A -85,B 0,C 180,E1 19348.811,E2 19348.811} C_VEL
LIN {X 0,Y 347.719,Z 1282.042,A -85,B 0,C 180,E1 19357.584,E2 19357.584} C_VEL
LIN {X 0,Y 349.892,Z 1265.47,A -85,B 0,C 180,E1 19367.223,E2 19367.223} C_VEL
LIN {X 0,Y 359.618,Z 1230.218,A -85,B 0,C 180,E1 19377.584,E2 19377.584} C_VEL
LIN {X 0,Y 390.219,Z 1163.761,A -85,B 0,C 180,E1 19389.617,E2 19389.617} C_VEL
LIN {X 0,Y 412.205,Z 1133.608,A -85,B 0,C 180,E1 19393.569,E2 19393.569} C_VEL
LIN {X 0,Y 381.36,Z 1187.672,A -85,B 0,C 180,E1 19402.442,E2 19402.442} C_VEL
LIN {X 0,Y 364.445,Z 1207.264,A -85,B 0,C 180,E1 19406.168,E2 19406.168} C_VEL
LIN {X 0,Y 347.566,Z 1233.699,A -85,B 0,C 180,E1 19417.229,E2 19417.229} C_VEL
LIN {X 0,Y 340.852,Z 1245.031,A -85,B 0,C 180,E1 19428.466,E2 19428.466} C_VEL
LIN {X 0,Y 339.738,Z 1243.934,A -85,B 0,C 180,E1 19438.745,E2 19438.745} C_VEL
LIN {X 0,Y 341.075,Z 1231.312,A -85,B 0,C 180,E1 19448.986,E2 19448.986} C_VEL
LIN {X 0,Y 346.698,Z 1205.226,A -85,B 0,C 180,E1 19459.194,E2 19459.194} C_VEL
LIN {X 0,Y 358.257,Z 1164.651,A -85,B 0,C 180,E1 19468.492,E2 19468.492} C_VEL
LIN {X 0,Y 372.703,Z 1112.974,A -85,B 0,C 180,E1 19475.75,E2 19475.75} C_VEL
LIN {X 0,Y 381.952,Z 1065.772,A -85,B 0,C 180,E1 19480.148,E2 19480.148} C_VEL
LIN {X 0,Y 362.889,Z 1008.022,A -85,B 0,C 180,E1 19486.298,E2 19486.298} C_VEL
LIN {X 0,Y 336.693,Z 948.94,A -85,B 0,C 180,E1 19492.815,E2 19492.815} C_VEL
LIN {X 0,Y 336.872,Z 950.236,A -85,B 0,C 180,E1 19494.536,E2 19494.536} C_VEL
LIN {X 0,Y 364.876,Z 1016.468,A -85,B 0,C 180,E1 19499.133,E2 19499.133} C_VEL
LIN {X 0,Y 367.433,Z 1039.87,A -85,B 0,C 180,E1 19499.927,E2 19499.927} C_VEL
LIN {X 0,Y 363.45,Z 1089.416,A -85,B 0,C 180,E1 19502.429,E2 19502.429} C_VEL
LIN {X 0,Y 355.852,Z 1132.649,A -85,B 0,C 180,E1 19507.204,E2 19507.204} C_VEL
LIN {X 0,Y 348.107,Z 1164.261,A -85,B 0,C 180,E1 19513.806,E2 19513.806} C_VEL
LIN {X 0,Y 343.539,Z 1181.691,A -85,B 0,C 180,E1 19521.044,E2 19521.044} C_VEL
LIN {X 0,Y 342.054,Z 1187.377,A -85,B 0,C 180,E1 19528.666,E2 19528.666} C_VEL
LIN {X 0,Y 343.805,Z 1179.482,A -85,B 0,C 180,E1 19537.545,E2 19537.545} C_VEL
LIN {X 0,Y 349.247,Z 1157.166,A -85,B 0,C 180,E1 19545.368,E2 19545.368} C_VEL
LIN {X 0,Y 356.678,Z 1122.028,A -85,B 0,C 180,E1 19551.624,E2 19551.624} C_VEL
LIN {X 0,Y 363.111,Z 1076.688,A -85,B 0,C 180,E1 19555.835,E2 19555.835} C_VEL
LIN {X 0,Y 365.829,Z 1026.882,A -85,B 0,C 180,E1 19557.76,E2 19557.76} C_VEL
LIN {X 0,Y 344.562,Z 966.532,A -85,B 0,C 180,E1 19561.2,E2 19561.2} C_VEL
LIN {X 0,Y 336.683,Z 948.94,A -85,B 0,C 180,E1 19562.661,E2 19562.661} C_VEL
LIN {X 0,Y 336.501,Z 948.94,A -85,B 0,C 180,E1 19575.607,E2 19575.607} C_VEL
LIN {X 0,Y 336.87,Z 948.94,A -85,B 0,C 180,E1 19586.318,E2 19586.318} C_VEL
LIN {X 0,Y 337.336,Z 948.94,A -85,B 0,C 180,E1 19597.487,E2 19597.487} C_VEL
LIN {X 0,Y 338.31,Z 948.94,A -85,B 0,C 180,E1 19608.327,E2 19608.327} C_VEL
LIN {X 0,Y 338.847,Z 948.94,A -85,B 0,C 180,E1 19618.692,E2 19618.692} C_VEL
LIN {X 0,Y 338.16,Z 948.94,A -85,B 0,C 180,E1 19629.013,E2 19629.013} C_VEL
LIN {X 0,Y 337.345,Z 948.94,A -85,B 0,C 180,E1 19639.694,E2 19639.694} C_VEL
LIN {X 0,Y 337.329,Z 950.839,A -85,B 0,C 180,E1 19648.52,E2 19648.52} C_VEL
LIN {X 0,Y 368.884,Z 1019.773,A -85,B 0,C 180,E1 19658.059,E2 19658.059} C_VEL
LIN {X 0,Y 388.221,Z 1074.149,A -85,B 0,C 180,E1 19664.676,E2 19664.676} C_VEL
LIN {X 0,Y 368.019,Z 1147.794,A -85,B 0,C 180,E1 19671.409,E2 19671.409} C_VEL
LIN {X 0,Y 352.195,Z 1206.99,A -85,B 0,C 180,E1 19680.148,E2 19680.148} C_VEL
LIN {X 0,Y 343.093,Z 1249.102,A -85,B 0,C 180,E1 19690.023,E2 19690.023} C_VEL
LIN {X 0,Y 340.209,Z 1273.832,A -85,B 0,C 180,E1 19699.818,E2 19699.818} C_VEL
LIN {X 0,Y 339.647,Z 1283.77,A -85,B 0,C 180,E1 19708.783,E2 19708.783} C_VEL
LIN {X 0,Y 339.728,Z 1281.651,A -85,B 0,C 180,E1 19717.764,E2 19717.764} C_VEL
LIN {X 0,Y 342.079,Z 1265.777,A -85,B 0,C 180,E1 19727.537,E2 19727.537} C_VEL
LIN {X 0,Y 352.404,Z 1232.011,A -85,B 0,C 180,E1 19738.053,E2 19738.053} C_VEL
LIN {X 0,Y 385.049,Z 1168.766,A -85,B 0,C 180,E1 19750.257,E2 19750.257} C_VEL
LIN {X 0,Y 403.96,Z 1144.983,A -85,B 0,C 180,E1 19753.624,E2 19753.624} C_VEL
LIN {X 0,Y 371.726,Z 1195.993,A -85,B 0,C 180,E1 19763.08,E2 19763.08} C_VEL
LIN {X 0,Y 364.445,Z 1207.264,A -85,B 0,C 180,E1 19766.168,E2 19766.168} C_VEL
LIN {X 0,Y 348.391,Z 1223.254,A -85,B 0,C 180,E1 19770.578,E2 19770.578} C_VEL
LIN {X 0,Y 336.341,Z 1240.893,A -85,B 0,C 180,E1 19781.292,E2 19781.292} C_VEL
LIN {X 0,Y 332.248,Z 1246.507,A -85,B 0,C 180,E1 19790.825,E2 19790.825} C_VEL
LIN {X 0,Y 331.802,Z 1242.214,A -85,B 0,C 180,E1 19801.336,E2 19801.336} C_VEL
LIN {X 0,Y 334.188,Z 1226.216,A -85,B 0,C 180,E1 19811.819,E2 19811.819} C_VEL
LIN {X 0,Y 342.22,Z 1194.535,A -85,B 0,C 180,E1 19822.518,E2 19822.518} C_VEL
LIN {X 0,Y 355.279,Z 1150.074,A -85,B 0,C 180,E1 19831.41,E2 19831.41} C_VEL
LIN {X 0,Y 370.229,Z 1094.905,A -85,B 0,C 180,E1 19838.164,E2 19838.164} C_VEL
LIN {X 0,Y 374.543,Z 1067.451,A -85,B 0,C 180,E1 19840.653,E2 19840.653} C_VEL
LIN {X 0,Y 355.656,Z 1009.836,A -85,B 0,C 180,E1 19846.977,E2 19846.977} C_VEL
LIN {X 0,Y 329.721,Z 952.824,A -85,B 0,C 180,E1 19853.71,E2 19853.71} C_VEL
LIN {X 0,Y 356.791,Z 1014.731,A -85,B 0,C 180,E1 19858.309,E2 19858.309} C_VEL
LIN {X 0,Y 360.638,Z 1036.02,A -85,B 0,C 180,E1 19859.178,E2 19859.178} C_VEL
LIN {X 0,Y 356.88,Z 1086.172,A -85,B 0,C 180,E1 19861.531,E2 19861.531} C_VEL
LIN {X 0,Y 349.436,Z 1129.474,A -85,B 0,C 180,E1 19866.091,E2 19866.091} C_VEL
LIN {X 0,Y 341.149,Z 1162.959,A -85,B 0,C 180,E1 19872.798,E2 19872.798} C_VEL
LIN {X 0,Y 335.696,Z 1182.622,A -85,B 0,C 180,E1 19880.833,E2 19880.833} C_VEL
LIN {X 0,Y 334.123,Z 1188.328,A -85,B 0,C 180,E1 19888.635,E2 19888.635} C_VEL
LIN {X 0,Y 335.946,Z 1180.457,A -85,B 0,C 180,E1 19897.723,E2 19897.723} C_VEL
LIN {X 0,Y 341.592,Z 1158.172,A -85,B 0,C 180,E1 19905.721,E2 19905.721} C_VEL
LIN {X 0,Y 349.334,Z 1123.066,A -85,B 0,C 180,E1 19912.102,E2 19912.102} C_VEL
LIN {X 0,Y 355.996,Z 1077.818,A -85,B 0,C 180,E1 19916.391,E2 19916.391} C_VEL
LIN {X 0,Y 358.716,Z 1025.443,A -85,B 0,C 180,E1 19918.426,E2 19918.426} C_VEL
LIN {X 0,Y 333.148,Z 959.421,A -85,B 0,C 180,E1 19922.642,E2 19922.642} C_VEL
LIN {X 0,Y 328.626,Z 948.94,A -85,B 0,C 180,E1 19923.766,E2 19923.766} C_VEL
LIN {X 0,Y 328.499,Z 948.94,A -85,B 0,C 180,E1 19935.625,E2 19935.625} C_VEL
LIN {X 0,Y 328.894,Z 948.94,A -85,B 0,C 180,E1 19948.464,E2 19948.464} C_VEL
LIN {X 0,Y 329.562,Z 948.94,A -85,B 0,C 180,E1 19960.503,E2 19960.503} C_VEL
LIN {X 0,Y 330.313,Z 948.94,A -85,B 0,C 180,E1 19970.719,E2 19970.719} C_VEL
LIN {X 0,Y 330.674,Z 948.94,A -85,B 0,C 180,E1 19981.289,E2 19981.289} C_VEL
LIN {X 0,Y 329.862,Z 948.94,A -85,B 0,C 180,E1 19991.924,E2 19991.924} C_VEL
LIN {X 0,Y 329.169,Z 948.94,A -85,B 0,C 180,E1 20003.047,E2 20003.047} C_VEL
LIN {X 0,Y 329.129,Z 950.357,A -85,B 0,C 180,E1 20007.137,E2 20007.137} C_VEL
LIN {X 0,Y 360.028,Z 1017.948,A -85,B 0,C 180,E1 20016.894,E2 20016.894} C_VEL
LIN {X 0,Y 381.009,Z 1075.418,A -85,B 0,C 180,E1 20024.167,E2 20024.167} C_VEL
LIN {X 0,Y 359.96,Z 1150.092,A -85,B 0,C 180,E1 20031.229,E2 20031.229} C_VEL
LIN {X 0,Y 344.212,Z 1207.46,A -85,B 0,C 180,E1 20039.979,E2 20039.979} C_VEL
LIN {X 0,Y 335.171,Z 1248.595,A -85,B 0,C 180,E1 20049.876,E2 20049.876} C_VEL
LIN {X 0,Y 332.234,Z 1273.369,A -85,B 0,C 180,E1 20059.921,E2 20059.921} C_VEL
LIN {X 0,Y 331.671,Z 1283.074,A -85,B 0,C 180,E1 20068.754,E2 20068.754} C_VEL
LIN {X 0,Y 331.729,Z 1281.279,A -85,B 0,C 180,E1 20077.952,E2 20077.952} C_VEL
LIN {X 0,Y 334.366,Z 1265.958,A -85,B 0,C 180,E1 20087.955,E2 20087.955} C_VEL
LIN {X 0,Y 346.791,Z 1230.441,A -85,B 0,C 180,E1 20099.41,E2 20099.41} C_VEL
LIN {X 0,Y 381.07,Z 1172.359,A -85,B 0,C 180,E1 20111.143,E2 20111.143} C_VEL
LIN {X 0,Y 395.729,Z 1155.438,A -85,B 0,C 180,E1 20113.703,E2 20113.703} C_VEL
LIN {X 0,Y 361.43,Z 1204.582,A -85,B 0,C 180,E1 20124.019,E2 20124.019} C_VEL
LIN {X 0,Y 348.391,Z 1223.254,A -85,B 0,C 180,E1 20130.578,E2 20130.578} C_VEL
LIN {X 0,Y 333.392,Z 1235.447,A -85,B 0,C 180,E1 20135.583,E2 20135.583} C_VEL
LIN {X 0,Y 325.112,Z 1246.599,A -85,B 0,C 180,E1 20147.899,E2 20147.899} C_VEL
LIN {X 0,Y 323.73,Z 1244.718,A -85,B 0,C 180,E1 20158.683,E2 20158.683} C_VEL
LIN {X 0,Y 325.201,Z 1231.486,A -85,B 0,C 180,E1 20169.428,E2 20169.428} C_VEL
LIN {X 0,Y 331.83,Z 1203.453,A -85,B 0,C 180,E1 20180.44,E2 20180.44} C_VEL
LIN {X 0,Y 344.539,Z 1161.002,A -85,B 0,C 180,E1 20190.102,E2 20190.102} C_VEL
LIN {X 0,Y 359.87,Z 1107.6,A -85,B 0,C 180,E1 20197.483,E2 20197.483} C_VEL
LIN {X 0,Y 367.535,Z 1070.622,A -85,B 0,C 180,E1 20200.985,E2 20200.985} C_VEL
LIN {X 0,Y 349.672,Z 1014.714,A -85,B 0,C 180,E1 20207.336,E2 20207.336} C_VEL
LIN {X 0,Y 326.916,Z 962.655,A -85,B 0,C 180,E1 20213.61,E2 20213.61} C_VEL
LIN {X 0,Y 352.285,Z 1023.724,A -85,B 0,C 180,E1 20218.065,E2 20218.065} C_VEL
LIN {X 0,Y 351.305,Z 1074.692,A -85,B 0,C 180,E1 20220.079,E2 20220.079} C_VEL
LIN {X 0,Y 344.478,Z 1119.924,A -85,B 0,C 180,E1 20224.149,E2 20224.149} C_VEL
LIN {X 0,Y 336.213,Z 1155.068,A -85,B 0,C 180,E1 20230.149,E2 20230.149} C_VEL
LIN {X 0,Y 329.308,Z 1178.941,A -85,B 0,C 180,E1 20237.967,E2 20237.967} C_VEL
LIN {X 0,Y 326.446,Z 1188.648,A -85,B 0,C 180,E1 20245.936,E2 20245.936} C_VEL
LIN {X 0,Y 326.621,Z 1186.754,A -85,B 0,C 180,E1 20253.93,E2 20253.93} C_VEL
LIN {X 0,Y 330.619,Z 1171.102,A -85,B 0,C 180,E1 20262.524,E2 20262.524} C_VEL
LIN {X 0,Y 338.116,Z 1141.305,A -85,B 0,C 180,E1 20269.941,E2 20269.941} C_VEL
LIN {X 0,Y 346.165,Z 1100.356,A -85,B 0,C 180,E1 20275.275,E2 20275.275} C_VEL
LIN {X 0,Y 351.193,Z 1052.328,A -85,B 0,C 180,E1 20278.332,E2 20278.332} C_VEL
LIN {X 0,Y 349.782,Z 1020.404,A -85,B 0,C 180,E1 20279.385,E2 20279.385} C_VEL
LIN {X 0,Y 324.181,Z 957.746,A -85,B 0,C 180,E1 20283.762,E2 20283.762} C_VEL
LIN {X 0,Y 320.498,Z 948.94,A -85,B 0,C 180,E1 20284.581,E2 20284.581} C_VEL
LIN {X 0,Y 320.468,Z 948.94,A -85,B 0,C 180,E1 20297.112,E2 20297.112} C_VEL
LIN {X 0,Y 320.674,Z 948.94,A -85,B 0,C 180,E1 20306.991,E2 20306.991} C_VEL
LIN {X 0,Y 321.368,Z 948.94,A -85,B 0,C 180,E1 20319.226,E2 20319.226} C_VEL
LIN {X 0,Y 322.33,Z 948.94,A -85,B 0,C 180,E1 20330.487,E2 20330.487} C_VEL
LIN {X 0,Y 322.699,Z 948.94,A -85,B 0,C 180,E1 20341.321,E2 20341.321} C_VEL
LIN {X 0,Y 321.805,Z 948.94,A -85,B 0,C 180,E1 20352.227,E2 20352.227} C_VEL
LIN {X 0,Y 320.991,Z 948.94,A -85,B 0,C 180,E1 20365.157,E2 20365.157} C_VEL
LIN {X 0,Y 352.771,Z 1019.768,A -85,B 0,C 180,E1 20376.201,E2 20376.201} C_VEL
LIN {X 0,Y 373.338,Z 1078.009,A -85,B 0,C 180,E1 20383.761,E2 20383.761} C_VEL
LIN {X 0,Y 352.196,Z 1151.206,A -85,B 0,C 180,E1 20390.904,E2 20390.904} C_VEL
LIN {X 0,Y 336.095,Z 1208.504,A -85,B 0,C 180,E1 20399.926,E2 20399.926} C_VEL
LIN {X 0,Y 327.062,Z 1249.149,A -85,B 0,C 180,E1 20410.063,E2 20410.063} C_VEL
LIN {X 0,Y 324.169,Z 1273.889,A -85,B 0,C 180,E1 20420.639,E2 20420.639} C_VEL
LIN {X 0,Y 323.725,Z 1282.327,A -85,B 0,C 180,E1 20428.723,E2 20428.723} C_VEL
LIN {X 0,Y 323.755,Z 1280.93,A -85,B 0,C 180,E1 20438.149,E2 20438.149} C_VEL
LIN {X 0,Y 327.103,Z 1264.813,A -85,B 0,C 180,E1 20449.016,E2 20449.016} C_VEL
LIN {X 0,Y 342.023,Z 1227.98,A -85,B 0,C 180,E1 20461.118,E2 20461.118} C_VEL
LIN {X 0,Y 377.23,Z 1176.028,A -85,B 0,C 180,E1 20472.042,E2 20472.042} C_VEL
LIN {X 0,Y 387.253,Z 1165.631,A -85,B 0,C 180,E1 20474.14,E2 20474.14} C_VEL
LIN {X 0,Y 355.294,Z 1207.035,A -85,B 0,C 180,E1 20483.298,E2 20483.298} C_VEL
LIN {X 0,Y 334.674,Z 1233.775,A -85,B 0,C 180,E1 20494.507,E2 20494.507} C_VEL
LIN {X 0,Y 333.392,Z 1235.447,A -85,B 0,C 180,E1 20495.583,E2 20495.583} C_VEL
LIN {X 0,Y 320.492,Z 1243.753,A -85,B 0,C 180,E1 20501.21,E2 20501.21} C_VEL
LIN {X 0,Y 315.822,Z 1247.583,A -85,B 0,C 180,E1 20513.127,E2 20513.127} C_VEL
LIN {X 0,Y 315.918,Z 1239.825,A -85,B 0,C 180,E1 20524.16,E2 20524.16} C_VEL
LIN {X 0,Y 319.827,Z 1219.643,A -85,B 0,C 180,E1 20535.158,E2 20535.158} C_VEL
LIN {X 0,Y 329.407,Z 1185.256,A -85,B 0,C 180,E1 20545.621,E2 20545.621} C_VEL
LIN {X 0,Y 344.425,Z 1137.145,A -85,B 0,C 180,E1 20554.406,E2 20554.406} C_VEL
LIN {X 0,Y 360.433,Z 1077.305,A -85,B 0,C 180,E1 20560.975,E2 20560.975} C_VEL
LIN {X 0,Y 345.719,Z 1025.256,A -85,B 0,C 180,E1 20567.052,E2 20567.052} C_VEL
LIN {X 0,Y 323.961,Z 972.251,A -85,B 0,C 180,E1 20573.482,E2 20573.482} C_VEL
LIN {X 0,Y 347.029,Z 1030.548,A -85,B 0,C 180,E1 20577.684,E2 20577.684} C_VEL
LIN {X 0,Y 343.71,Z 1082.31,A -85,B 0,C 180,E1 20579.878,E2 20579.878} C_VEL
LIN {X 0,Y 335.99,Z 1126.705,A -85,B 0,C 180,E1 20584.346,E2 20584.346} C_VEL
LIN {X 0,Y 327.16,Z 1161.214,A -85,B 0,C 180,E1 20590.987,E2 20590.987} C_VEL
LIN {X 0,Y 320.768,Z 1182.351,A -85,B 0,C 180,E1 20599.026,E2 20599.026} C_VEL
LIN {X 0,Y 318.261,Z 1190.23,A -85,B 0,C 180,E1 20608.567,E2 20608.567} C_VEL
LIN {X 0,Y 320.232,Z 1182.407,A -85,B 0,C 180,E1 20618.104,E2 20618.104} C_VEL
LIN {X 0,Y 326.34,Z 1160.182,A -85,B 0,C 180,E1 20626.477,E2 20626.477} C_VEL
LIN {X 0,Y 334.723,Z 1125.141,A -85,B 0,C 180,E1 20633.121,E2 20633.121} C_VEL
LIN {X 0,Y 341.769,Z 1081.137,A -85,B 0,C 180,E1 20637.498,E2 20637.498} C_VEL
LIN {X 0,Y 344.88,Z 1028.982,A -85,B 0,C 180,E1 20639.665,E2 20639.665} C_VEL
LIN {X 0,Y 320.901,Z 967.061,A -85,B 0,C 180,E1 20643.923,E2 20643.923} C_VEL
LIN {X 0,Y 312.397,Z 948.94,A -85,B 0,C 180,E1 20645.829,E2 20645.829} C_VEL
LIN {X 0,Y 312.354,Z 948.94,A -85,B 0,C 180,E1 20658.969,E2 20658.969} C_VEL
LIN {X 0,Y 312.711,Z 948.94,A -85,B 0,C 180,E1 20669.329,E2 20669.329} C_VEL
LIN {X 0,Y 313.563,Z 948.94,A -85,B 0,C 180,E1 20681.633,E2 20681.633} C_VEL
LIN {X 0,Y 314.379,Z 948.94,A -85,B 0,C 180,E1 20693.04,E2 20693.04} C_VEL
LIN {X 0,Y 314.63,Z 948.94,A -85,B 0,C 180,E1 20704.122,E2 20704.122} C_VEL
LIN {X 0,Y 313.56,Z 948.94,A -85,B 0,C 180,E1 20715.412,E2 20715.412} C_VEL
LIN {X 0,Y 313.106,Z 950.091,A -85,B 0,C 180,E1 20724.303,E2 20724.303} C_VEL
LIN {X 0,Y 344.001,Z 1017.936,A -85,B 0,C 180,E1 20734.971,E2 20734.971} C_VEL
LIN {X 0,Y 365.998,Z 1079.512,A -85,B 0,C 180,E1 20743.267,E2 20743.267} C_VEL
LIN {X 0,Y 344.056,Z 1153.551,A -85,B 0,C 180,E1 20750.74,E2 20750.74} C_VEL
LIN {X 0,Y 327.589,Z 1211.109,A -85,B 0,C 180,E1 20760.214,E2 20760.214} C_VEL
LIN {X 0,Y 318.804,Z 1250.638,A -85,B 0,C 180,E1 20770.611,E2 20770.611} C_VEL
LIN {X 0,Y 316.136,Z 1273.892,A -85,B 0,C 180,E1 20781.095,E2 20781.095} C_VEL
LIN {X 0,Y 315.776,Z 1281.564,A -85,B 0,C 180,E1 20788.691,E2 20788.691} C_VEL
LIN {X 0,Y 315.68,Z 1281.435,A -85,B 0,C 180,E1 20796.97,E2 20796.97} C_VEL
LIN {X 0,Y 318.483,Z 1267.855,A -85,B 0,C 180,E1 20808.11,E2 20808.11} C_VEL
LIN {X 0,Y 332.861,Z 1234.456,A -85,B 0,C 180,E1 20820.546,E2 20820.546} C_VEL
LIN {X 0,Y 369.482,Z 1183.889,A -85,B 0,C 180,E1 20832.212,E2 20832.212} C_VEL
LIN {X 0,Y 378.809,Z 1174.741,A -85,B 0,C 180,E1 20834.216,E2 20834.216} C_VEL
LIN {X 0,Y 345.152,Z 1214.388,A -85,B 0,C 180,E1 20844.161,E2 20844.161} C_VEL
LIN {X 0,Y 324.474,Z 1238.936,A -85,B 0,C 180,E1 20856.6,E2 20856.6} C_VEL
LIN {X 0,Y 320.492,Z 1243.753,A -85,B 0,C 180,E1 20861.21,E2 20861.21} C_VEL
LIN {X 0,Y 309.368,Z 1248.117,A -85,B 0,C 180,E1 20867.294,E2 20867.294} C_VEL
LIN {X 0,Y 307.802,Z 1244.366,A -85,B 0,C 180,E1 20880.028,E2 20880.028} C_VEL
LIN {X 0,Y 310.043,Z 1228.081,A -85,B 0,C 180,E1 20891.68,E2 20891.68} C_VEL
LIN {X 0,Y 318.565,Z 1196.449,A -85,B 0,C 180,E1 20903.175,E2 20903.175} C_VEL
LIN {X 0,Y 332.872,Z 1151.097,A -85,B 0,C 180,E1 20912.812,E2 20912.812} C_VEL
LIN {X 0,Y 348.907,Z 1095.939,A -85,B 0,C 180,E1 20919.9,E2 20919.9} C_VEL
LIN {X 0,Y 352.832,Z 1074.362,A -85,B 0,C 180,E1 20921.985,E2 20921.985} C_VEL
LIN {X 0,Y 335.358,Z 1018.645,A -85,B 0,C 180,E1 20928.716,E2 20928.716} C_VEL
LIN {X 0,Y 320.76,Z 981.963,A -85,B 0,C 180,E1 20933.322,E2 20933.322} C_VEL
LIN {X 0,Y 340.313,Z 1033.941,A -85,B 0,C 180,E1 20937.045,E2 20937.045} C_VEL
LIN {X 0,Y 336.739,Z 1084.204,A -85,B 0,C 180,E1 20939.281,E2 20939.281} C_VEL
LIN {X 0,Y 328.592,Z 1128.67,A -85,B 0,C 180,E1 20943.909,E2 20943.909} C_VEL
LIN {X 0,Y 319.654,Z 1162.109,A -85,B 0,C 180,E1 20950.523,E2 20950.523} C_VEL
LIN {X 0,Y 312.982,Z 1183.278,A -85,B 0,C 180,E1 20958.749,E2 20958.749} C_VEL
LIN {X 0,Y 310.333,Z 1191.181,A -85,B 0,C 180,E1 20968.53,E2 20968.53} C_VEL
LIN {X 0,Y 312.395,Z 1183.38,A -85,B 0,C 180,E1 20978.309,E2 20978.309} C_VEL
LIN {X 0,Y 318.744,Z 1161.186,A -85,B 0,C 180,E1 20986.881,E2 20986.881} C_VEL
LIN {X 0,Y 327.459,Z 1126.178,A -85,B 0,C 180,E1 20993.665,E2 20993.665} C_VEL
LIN {X 0,Y 334.795,Z 1082.017,A -85,B 0,C 180,E1 20998.141,E2 20998.141} C_VEL
LIN {X 0,Y 337.86,Z 1030.216,A -85,B 0,C 180,E1 21000.353,E2 21000.353} C_VEL
LIN {X 0,Y 313.744,Z 968.4,A -85,B 0,C 180,E1 21004.815,E2 21004.815} C_VEL
LIN {X 0,Y 304.346,Z 948.94,A -85,B 0,C 180,E1 21006.991,E2 21006.991} C_VEL
LIN {X 0,Y 304.271,Z 948.94,A -85,B 0,C 180,E1 21020.506,E2 21020.506} C_VEL
LIN {X 0,Y 304.763,Z 948.94,A -85,B 0,C 180,E1 21031.731,E2 21031.731} C_VEL
LIN {X 0,Y 305.934,Z 948.94,A -85,B 0,C 180,E1 21044.987,E2 21044.987} C_VEL
LIN {X 0,Y 306.657,Z 948.94,A -85,B 0,C 180,E1 21056.695,E2 21056.695} C_VEL
LIN {X 0,Y 306.331,Z 948.94,A -85,B 0,C 180,E1 21067.087,E2 21067.087} C_VEL
LIN {X 0,Y 305.25,Z 948.94,A -85,B 0,C 180,E1 21078.827,E2 21078.827} C_VEL
LIN {X 0,Y 305.206,Z 949.874,A -85,B 0,C 180,E1 21082.805,E2 21082.805} C_VEL
LIN {X 0,Y 336.07,Z 1018.342,A -85,B 0,C 180,E1 21094.008,E2 21094.008} C_VEL
LIN {X 0,Y 358.418,Z 1081.747,A -85,B 0,C 180,E1 21102.82,E2 21102.82} C_VEL
LIN {X 0,Y 336.071,Z 1155.059,A -85,B 0,C 180,E1 21110.466,E2 21110.466} C_VEL
LIN {X 0,Y 319.464,Z 1211.981,A -85,B 0,C 180,E1 21120.164,E2 21120.164} C_VEL
LIN {X 0,Y 310.677,Z 1251.042,A -85,B 0,C 180,E1 21130.825,E2 21130.825} C_VEL
LIN {X 0,Y 308.14,Z 1273.807,A -85,B 0,C 180,E1 21141.576,E2 21141.576} C_VEL
LIN {X 0,Y 307.948,Z 1281.871,A -85,B 0,C 180,E1 21151.481,E2 21151.481} C_VEL
LIN {X 0,Y 308.154,Z 1277.863,A -85,B 0,C 180,E1 21161.43,E2 21161.43} C_VEL
LIN {X 0,Y 314.99,Z 1257.969,A -85,B 0,C 180,E1 21173.46,E2 21173.46} C_VEL
